   // sequencer 1
   INITIAL_STEP Initialschritt:   // S1, max time T#10S, warning time T#7S
              N    #sq.init
              R    #sq.inHoming
              R    #sq.running
              R    #sq.done
              R    "FG01Actors".Lasermarker.setWorkPos
              R    #qxNok
              R    "FG01Actors".Camera.setTrigger
   END_STEP
   TRANSITION Automatikablauf FROM Initialschritt TO Grundstellung   // T1
      := NOT #signals.isHoming;
   END_TRANSITION
   TRANSITION Grundstellungsfahrt FROM Initialschritt TO "Start Grundstellungsfahrt"   // T5
      := #signals.isHoming;
   END_TRANSITION
   STEP Grundstellung:   // S2, max time T#10S, warning time T#7S
              N    #sq.isWaiting
              N    "FG01Globals".SQ1.readyForIndex
   END_STEP
   TRANSITION Freigabe FROM Grundstellung TO SK_läuft   // T2
      := #sq.inHome AND NOT #signals.isInAutoStoping AND #sq.start AND NOT #sq.done AND #signals.releaseNextJog;
   END_TRANSITION
   STEP SK_läuft:   // S3, max time T#10S, warning time T#7S
              S    #sq.running
   END_STEP
   TRANSITION Trans3 FROM SK_läuft TO ReaderWindowToWork   // T3
      := "AlwaysTRUE";
   END_TRANSITION
   STEP Fertigmeldung:   // S4, max time T#10S, warning time T#7S
              R    #sq.running
              S    #sq.done
   END_STEP
   TRANSITION Fertig FROM Fertigmeldung TO Ende   // T4
      := "AlwaysTRUE";
   END_TRANSITION
   STEP "Start Grundstellungsfahrt":   // S5, max time T#10S, warning time T#7S
              S    #sq.inHoming
   END_STEP
   TRANSITION GST_Aktiv FROM "Start Grundstellungsfahrt" TO GS_GripperHome   // T6
      := #signals.releaseCycle;
   END_TRANSITION
   STEP "Fertig Grundstellungsfahrt":   // S6, max time T#10S, warning time T#7S
              R    #sq.inHoming
   END_STEP
   TRANSITION GST_Beendet FROM "Fertig Grundstellungsfahrt" TO Ende   // T7
      := "AlwaysTRUE";
   END_TRANSITION
   STEP Ende:   // S7, max time T#10S, warning time T#7S
   END_STEP
   TRANSITION Beendet FROM Ende TO Grundstellung   // T8, jump
      := "AlwaysTRUE";
   END_TRANSITION
   STEP ResetRelease:   // S8, max time T#10S, warning time T#7S
      supervision V := (#ResetRelease.U >= t#10s) AND NOT #DoneToIndexer.TT AND #signals.releaseCycle;
          S1  R    "TransportGlobals".Index01.release
   END_STEP
   TRANSITION DoneToIndexer FROM ResetRelease TO JogS7   // T9
      := true;
   END_TRANSITION
   STEP GS_GripperHome:   // S14, max time T#10S, warning time T#7S
      supervision V := #sstReleaseCycle.T >= #itMaxRuntime;
              R    "FG01Actors".Gripper.setWorkPos
              S    "FG01Actors".Gripper.setHomePos
   END_STEP
   TRANSITION GS_GripperInHome FROM GS_GripperHome TO GS_PlattformHome   // T15
      := "FG01Actors".Gripper.inHomePos;
   END_TRANSITION
   STEP GS_PlattformHome:   // S15, max time T#10S, warning time T#7S
      supervision V := #sstReleaseCycle.T >= #itMaxRuntime;
              S    "FG01Actors".Plattform.setHomePos
              R    "FG01Actors".Plattform.setWorkPos
   END_STEP
   TRANSITION GS_PlattformInHome FROM GS_PlattformHome TO GS_ReaderWindowHome   // T16
      := "FG01Actors".Plattform.inHomePos;
   END_TRANSITION
   STEP GS_ReaderWindowHome:   // S16, max time T#10S, warning time T#7S
      supervision V := #sstReleaseCycle.T >= #itMaxRuntime;
              R    "FG01Actors".ReaderWindow.setWorkPos
              S    "FG01Actors".ReaderWindow.setHomePos
   END_STEP
   TRANSITION GS_ReaderWindowInHome FROM GS_ReaderWindowHome TO GS_OpenGates   // T17
      := "FG01Actors".ReaderWindow.inHomePos;
   END_TRANSITION
   STEP PlattformToWork:   // S17, max time T#10S, warning time T#7S
      supervision V := #sstReleaseCycle.T >= #itMaxRuntime;
              R    "FG01Actors".Plattform.setHomePos
              S    "FG01Actors".Plattform.setWorkPos
   END_STEP
   TRANSITION PlattformIsInWork FROM PlattformToWork TO JogS4   // T18
      := "FG01Actors".Plattform.inWorkPos;
   END_TRANSITION
   STEP ReaderWindowToWork:   // S18, max time T#10S, warning time T#7S
      supervision V := #sstReleaseCycle.T >= #itMaxRuntime;
              S    "FG01Actors".ReaderWindow.setWorkPos
              R    "FG01Actors".ReaderWindow.setHomePos
   END_STEP
   TRANSITION ReaderWindowInWork FROM ReaderWindowToWork TO JogS1   // T19
      := "FG01Actors".ReaderWindow.inWorkPos;
   END_TRANSITION
   STEP GripperToWork:   // S19, max time T#10S, warning time T#7S
      supervision V := #sstReleaseCycle.T >= #itMaxRuntime;
              S    "FG01Actors".Gripper.setWorkPos
              R    "FG01Actors".Gripper.setHomePos
   END_STEP
   TRANSITION GripperInWork FROM GripperToWork TO JogS3   // T20
      := "FG01Actors".Gripper.inWorkPos;
   END_TRANSITION
   STEP GripperToHome:   // S20, max time T#10S, warning time T#7S
      supervision V := #sstReleaseCycle.T >= #itMaxRuntime;
              R    "FG01Actors".Gripper.setWorkPos
              S    "FG01Actors".Gripper.setHomePos
   END_STEP
   TRANSITION GripperInHome FROM GripperToHome TO JogS9   // T21
      := "FG01Actors".Gripper.inHomePos;
   END_TRANSITION
   STEP PlattformToHome:   // S21, max time T#10S, warning time T#7S
      supervision V := #sstReleaseCycle.T >= #itMaxRuntime;
              S    "FG01Actors".Plattform.setHomePos
              R    "FG01Actors".Plattform.setWorkPos
   END_STEP
   TRANSITION PlattformIsInWork_1 FROM PlattformToHome TO JogS8   // T22
      := "FG01Actors".Plattform.inHomePos;
   END_TRANSITION
   STEP JogS3:   // S28, max time T#10S, warning time T#7S
              N    #sq.jogDone
   END_STEP
   TRANSITION JogT3 FROM JogS3 TO PlattformToWork   // T30
      := #signals.releaseNextJog;
   END_TRANSITION
   STEP JogS4:   // S29, max time T#10S, warning time T#7S
              N    #sq.jogDone
   END_STEP
   TRANSITION JogT4 FROM JogS4 TO CheckLaserOn   // T31
      := #signals.releaseNextJog;
   END_TRANSITION
   STEP JogS1:   // S30, max time T#10S, warning time T#7S
              N    #sq.jogDone
   END_STEP
   TRANSITION JogT1 FROM JogS1 TO Set_Trigger   // T32
      := #signals.releaseNextJog;
   END_TRANSITION
   STEP JogS7:   // S31, max time T#10S, warning time T#7S
              N    #sq.jogDone
   END_STEP
   TRANSITION JogT7 FROM JogS7 TO PlattformToHome   // T33
      := #signals.releaseNextJog;
   END_TRANSITION
   STEP Laser:   // S32, max time T#10S, warning time T#7S
      supervision V := #sstReleaseCycle.T >= #itMaxRuntime;
              N    "FG01Actors".Lasermarker.setWorkPos
   END_STEP
   TRANSITION LaserDone FROM Laser TO JogS6   // T34
      := (#Laser.T >= t#3s) AND "FG01Actors".Lasermarker.workAct;
   END_TRANSITION
   STEP JogS8:   // S33, max time T#10S, warning time T#7S
              N    #sq.jogDone
   END_STEP
   TRANSITION JogT8 FROM JogS8 TO GripperToHome   // T35
      := #signals.releaseNextJog;
   END_TRANSITION
   STEP ReaderWindowToHome:   // S22, max time T#10S, warning time T#7S
      supervision V := #sstReleaseCycle.T >= #itMaxRuntime;
              R    "FG01Actors".ReaderWindow.setWorkPos
              S    "FG01Actors".ReaderWindow.setHomePos
   END_STEP
   TRANSITION ReaderWindowInHome FROM ReaderWindowToHome TO Fertigmeldung   // T23
      := "FG01Actors".ReaderWindow.inHomePos;
   END_TRANSITION
   STEP CloseGates:   // S34, max time T#10S, warning time T#7S
      supervision V := #sstReleaseCycle.T >= #itMaxRuntime;
              S    "FG01Actors".Gate_1.setWorkPos
              S    "FG01Actors".Gate_2.setWorkPos
   END_STEP
   TRANSITION GatesClosed FROM CloseGates TO JogS5   // T36
      := "FG01Actors".Gate_1.inWorkPos AND "FG01Actors".Gate_2.inWorkPos;
   END_TRANSITION
   STEP JogS5:   // S35, max time T#10S, warning time T#7S
              N    #sq.jogDone
   END_STEP
   TRANSITION JogT5 FROM JogS5 TO Laser   // T37
      := #signals.releaseNextJog;
   END_TRANSITION
   STEP JogS9:   // S36, max time T#10S, warning time T#7S
              N    #sq.jogDone
   END_STEP
   TRANSITION JogT9 FROM JogS9 TO ReaderWindowToHome   // T38
      := #signals.releaseNextJog;
   END_TRANSITION
   STEP OpenGates:   // S37, max time T#10S, warning time T#7S
      supervision V := #sstReleaseCycle.T >= #itMaxRuntime;
              R    "FG01Actors".Gate_1.setWorkPos
              R    "FG01Actors".Gate_2.setWorkPos
   END_STEP
   TRANSITION GatesOpened FROM OpenGates TO ResetRelease   // T39
      := "FG01Actors".Gate_1.inHomePos AND "FG01Actors".Gate_2.inHomePos;
   END_TRANSITION
   STEP JogS6:   // S38, max time T#10S, warning time T#7S
              N    #sq.jogDone
   END_STEP
   TRANSITION JogT6 FROM JogS6 TO OpenGates   // T40
      := #signals.releaseNextJog;
   END_TRANSITION
   STEP GS_OpenGates:   // S39, max time T#10S, warning time T#7S
      supervision V := #sstReleaseCycle.T >= #itMaxRuntime;
              R    "FG01Actors".Gate_1.setWorkPos
              R    "FG01Actors".Gate_2.setWorkPos
   END_STEP
   TRANSITION GS_GatesOpened FROM GS_OpenGates TO "Fertig Grundstellungsfahrt"   // T41
      := "FG01Actors".Gate_1.inHomePos AND "FG01Actors".Gate_2.inHomePos;
   END_TRANSITION
   STEP CheckLaserOn:   // S40, max time T#10S, warning time T#7S
   END_STEP
   TRANSITION LaserIsOn FROM CheckLaserOn TO CloseGates   // T42
      := "FG01Globals".laserOn;
   END_TRANSITION
   TRANSITION LaserIsOff FROM CheckLaserOn TO ResetRelease   // T43
      := NOT "FG01Globals".laserOn;
   END_TRANSITION
   STEP Set_Trigger:   // S9, max time T#10S, warning time T#7S
      supervision V := #sstReleaseCycle.T >= #itMaxRuntime;
              S    "FG01Actors".Camera.setTrigger
   END_STEP
   TRANSITION TriggerIsSet FROM Set_Trigger TO Wait_Busy_Done   // T10
      := "FG01Actors".Camera.isBusy;
   END_TRANSITION
   STEP Wait_Busy_Done:   // S11, max time T#10S, warning time T#7S
      supervision V := #sstReleaseCycle.T >= #itMaxRuntime;
   END_STEP
   TRANSITION CamIsDone FROM Wait_Busy_Done TO Check_Result   // T12
      := NOT "FG01Actors".Camera.isBusy;
   END_TRANSITION
   STEP Reset_Trigger:   // S12, max time T#10S, warning time T#7S
      supervision V := #sstReleaseCycle.T >= #itMaxRuntime;
              R    "FG01Actors".Camera.setTrigger
   END_STEP
   TRANSITION TriggerIsReseted FROM Reset_Trigger TO JogS2   // T13
      := "FG01Actors".Camera.isReady;
   END_TRANSITION
   STEP JogS2:   // S41, max time T#10S, warning time T#7S
              N    #sq.jogDone
   END_STEP
   TRANSITION JogT2 FROM JogS2 TO GripperToWork   // T44
      := #signals.releaseNextJog;
   END_TRANSITION
   STEP Check_Result:   // S42, max time T#10S, warning time T#7S
      supervision V := #sstReleaseCycle.T >= #itMaxRuntime;
   END_STEP
   TRANSITION "Result Ok" FROM Check_Result TO Reset_Trigger   // T45
      := "FG01Actors".Camera.resultOk;
   END_TRANSITION
   TRANSITION "Result Nok" FROM Check_Result TO NIO   // T46
      := "FG01Actors".Camera.resultNok;
   END_TRANSITION
   STEP NIO:   // S43, max time T#10S, warning time T#7S
          S1  S    #qxNok
              R    "FG01Actors".Camera.setTrigger
   END_STEP
   TRANSITION NIO_Quittiert FROM NIO TO Reset_Trigger   // T47
      := NOT #qxNok;
   END_TRANSITION

   // permanent post-instructions
   NETWORK 1
   TITLE = Störungssignal weitergeben / Forward fault signal
      #sq.error := #ERR_FLT;
   NETWORK 2
   TITLE = Ablauf ist aktiv / Sequence active
      #qxIsActive := #sq.running;
   NETWORK 3
   TITLE = steht in Grundstellung / in home position
      #qxIsInHome := #sq.inHome AND NOT #sq.running;
   NETWORK 4
   TITLE = NIO-Erkennung zurücksetzen / Reset NOK detection
      IF #signals.ack THEN #qxNok := FALSE; END_IF;
END_FUNCTION_BLOCK

FUNCTION "FG01StepSequences" : Void   // FC1110, FBD
TITLE = Schrittkettensteuerung / Sequence control
{ S7_Optimized_Access := 'TRUE' }
VERSION : 0.1
// Ersteller: Andreas Fast Automation
// Kontakt per LinkedIn: https://www.linkedin.com/in/automation-fast-andreas/
// 
// Das Projekt dient zu Demonstrationszwecken und kann frei genutzt werden.
// 
// Bausteinbeschreibung:
// Author: Andreas Fast Automation
// Kontakt per LinkedIn: https://www.linkedin.com/in/automation-fast-andreas/
// 
// This project is intended for demonstration purposes and may be used freely.
// 
// Block description:
   VAR_IN_OUT
      station : "typeStation";
   END_VAR
   VAR_TEMP
      tempInit : Bool;
      tempAck : Bool;
      tempSwAuto : Bool;
      tempSwMan : Bool;
      tempSwTap : Bool;
      tempPush : Bool;
   END_VAR
BEGIN

REGION Network 1: GRAPH-Parameter / GRAPH parameters
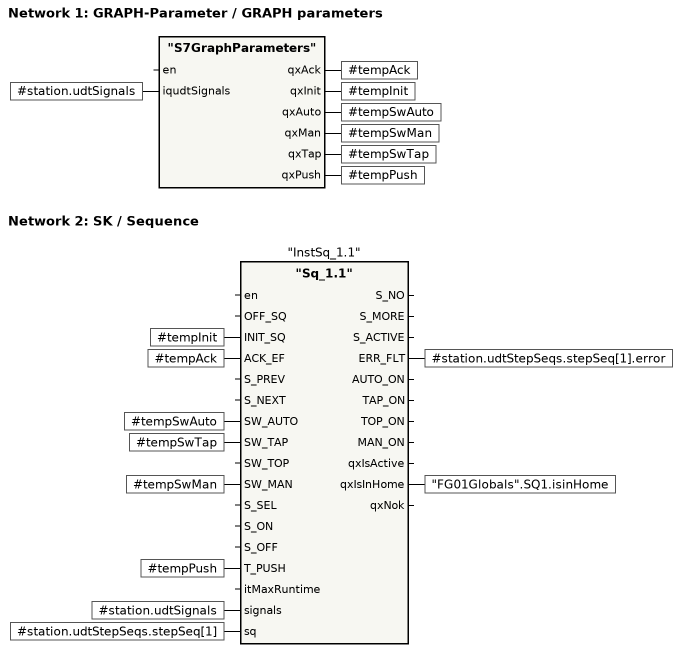
   "S7GraphParameters"(iqudtSignals := #station.udtSignals,
                       qxAck => #tempAck,
                       qxInit => #tempInit,
                       qxAuto => #tempSwAuto,
                       qxMan => #tempSwMan,
                       qxTap => #tempSwTap,
                       qxPush => #tempPush);
END_REGION

REGION Network 2: SK / Sequence
   "InstSq_1.1"(INIT_SQ := #tempInit,   // "Sq_1.1"
                ACK_EF := #tempAck,
                SW_AUTO := #tempSwAuto,
                SW_TAP := #tempSwTap,
                SW_MAN := #tempSwMan,
                T_PUSH := #tempPush,
                signals := #station.udtSignals,
                sq := #station.udtStepSeqs.stepSeq[1],
                ERR_FLT => #station.udtStepSeqs.stepSeq[1].error,
                qxIsInHome => "FG01Globals".SQ1.isinHome);
END_REGION
END_FUNCTION

// folder: 2. Machine/02_FG02

FUNCTION_BLOCK "FG02Control"   // FB1200, FBD
TITLE = Station 2 Hauptaufruf / Station 2 main call
{ S7_Optimized_Access := 'TRUE' }
VERSION : 0.1
// Ersteller: Andreas Fast Automation
// Kontakt per LinkedIn: https://www.linkedin.com/in/automation-fast-andreas/
// 
// Das Projekt dient zu Demonstrationszwecken und kann frei genutzt werden.
// 
// Bausteinbeschreibung:
// Author: Andreas Fast Automation
// Kontakt per LinkedIn: https://www.linkedin.com/in/automation-fast-andreas/
// 
// This project is intended for demonstration purposes and may be used freely.
// 
// Block description:
   VAR_INPUT
      stationNo : Int := 2;   // Stationsnummer / Station number
   END_VAR
   VAR_IN_OUT
      machine : "typeMachine";
      station : "typeStation";
      manualMovement : "typeManualMovements";
      plcErrMsg : "typePlcErrMsg";
      hmiErrMsg : "typeHmiErrMsg";
   END_VAR
   VAR
      instStationControl : "StationControl";
      instActorControl : "FG02ActorControl";
      instStationState : "StationState";
      sinstStationCycleTime : "StationCycleTime";
   END_VAR
BEGIN

REGION Network 1: Stationssteuerung / Station control
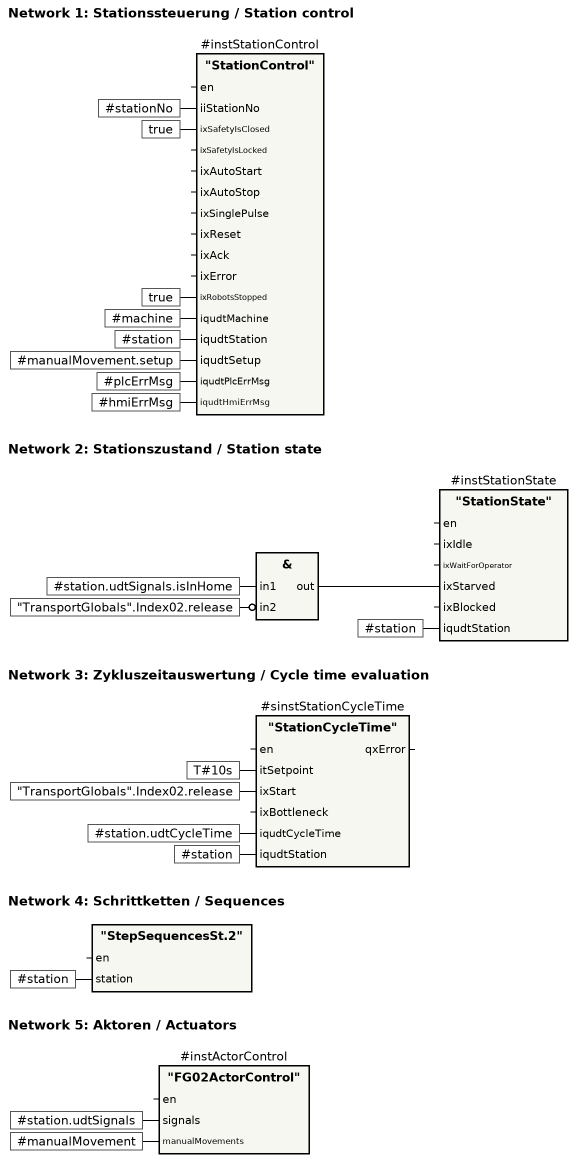
   #instStationControl(iiStationNo := #stationNo,   // "StationControl"
                       ixSafetyIsClosed := true,
                       ixRobotsStopped := true,
                       iqudtMachine := #machine,
                       iqudtStation := #station,
                       iqudtSetup := #manualMovement.setup,
                       iqudtPlcErrMsg := #plcErrMsg,
                       iqudtHmiErrMsg := #hmiErrMsg);
END_REGION

REGION Network 2: Stationszustand / Station state
   #instStationState(ixStarved := #station.udtSignals.isInHome AND NOT "TransportGlobals".Index02.release,   // "StationState"
                     iqudtStation := #station);
END_REGION

REGION Network 3: Zykluszeitauswertung / Cycle time evaluation
   #sinstStationCycleTime(itSetpoint := T#10s,   // "StationCycleTime"
                          ixStart := "TransportGlobals".Index02.release,
                          iqudtCycleTime := #station.udtCycleTime,
                          iqudtStation := #station);
END_REGION

REGION Network 4: Schrittketten / Sequences
   "StepSequencesSt.2"(station := #station);
END_REGION

REGION Network 5: Aktoren / Actuators
   #instActorControl(signals := #station.udtSignals, manualMovements := #manualMovement);   // "FG02ActorControl"
END_REGION
END_FUNCTION_BLOCK

FUNCTION_BLOCK "FG02ActorControl"   // FB1202, FBD
TITLE = Aktoransteuerung / Actuator control
{ S7_Optimized_Access := 'TRUE' }
VERSION : 0.1
// Ersteller: Andreas Fast Automation
// Kontakt per LinkedIn: https://www.linkedin.com/in/automation-fast-andreas/
// 
// Das Projekt dient zu Demonstrationszwecken und kann frei genutzt werden.
// 
// Bausteinbeschreibung:
// Author: Andreas Fast Automation
// Kontakt per LinkedIn: https://www.linkedin.com/in/automation-fast-andreas/
// 
// This project is intended for demonstration purposes and may be used freely.
// 
// Block description:
   VAR_IN_OUT
      signals : "typeStationSignals";
      manualMovements : "typeManualMovements";
   END_VAR
   VAR
      instCamera : "Actor_1Out_SimpleCamera";
      instActorReserved3 : "Actor_Reserved";
      instActorReserved4 : "Actor_Reserved";
   END_VAR
BEGIN

REGION Network 1: Kamera / Camera
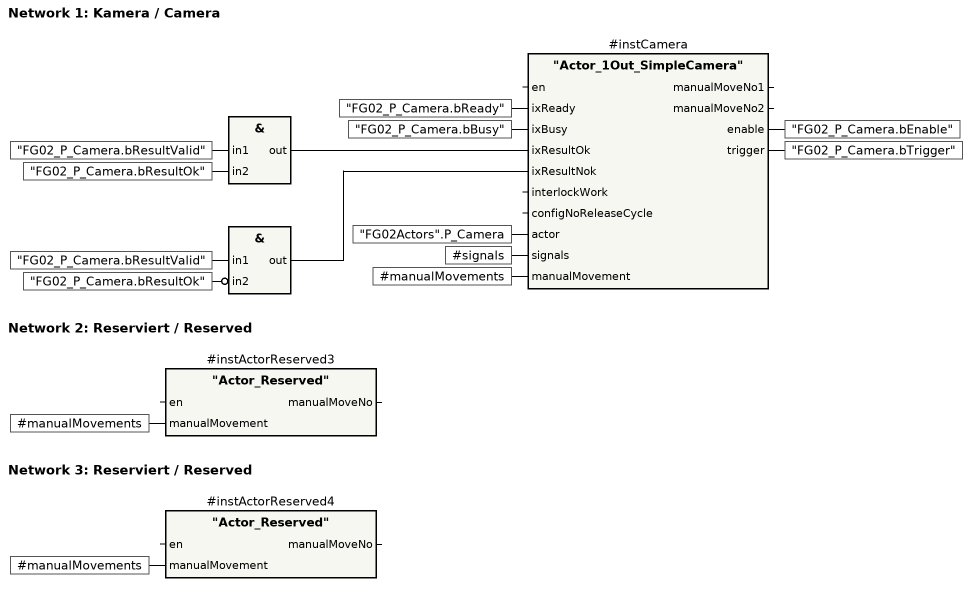
   #instCamera(ixReady := "FG02_P_Camera.bReady",   // "Actor_1Out_SimpleCamera"
               ixBusy := "FG02_P_Camera.bBusy",
               ixResultOk := "FG02_P_Camera.bResultValid" AND "FG02_P_Camera.bResultOk",
               ixResultNok := "FG02_P_Camera.bResultValid" AND NOT "FG02_P_Camera.bResultOk",
               actor := "FG02Actors".P_Camera,
               signals := #signals,
               manualMovement := #manualMovements,
               enable => "FG02_P_Camera.bEnable",
               trigger => "FG02_P_Camera.bTrigger");
END_REGION

REGION Network 2: Reserviert / Reserved
   #instActorReserved3(manualMovement := #manualMovements);   // "Actor_Reserved"
END_REGION

REGION Network 3: Reserviert / Reserved
   #instActorReserved4(manualMovement := #manualMovements);   // "Actor_Reserved"
END_REGION
END_FUNCTION_BLOCK

// folder: 2. Machine/02_FG02/Stepsequences

FUNCTION_BLOCK "Sq_2.1"   // FB1211, GRAPH_PLUS
{ S7_Optimized_Access := 'TRUE' }
VERSION : 0.1
   VAR_INPUT
      OFF_SQ : Bool := false;   // Kette ausschalten
      INIT_SQ : Bool := false;   // Kette in Initialzustand versetzen
      ACK_EF : Bool := false;   // Alle Fehler und Störungen quittieren
      S_PREV : Bool := false;   // Vorherigen Schritt am Parameter S_NO ausgeben
      S_NEXT : Bool := false;   // Nächsten Schritt am Parameter S_NO anzeigen
      SW_AUTO : Bool := false;   // Automatischer Betrieb
      SW_TAP : Bool := false;   // Halbautomatisch/Weiterschalten mit Transition
      SW_TOP : Bool := false;   // Halbautomatisch/Ignoriere Transition
      SW_MAN : Bool := false;   // Handbetrieb
      S_SEL : Int := 0;   // Schritt auswählen, der an S_NO ausgegeben werden soll
      S_ON : Bool := false;   // Schritt aktivieren, der an Parameter S_NO anliegt
      S_OFF : Bool := false;   // Schritt deaktivieren, der an Parameter S_NO anliegt
      T_PUSH : Bool := false;   // Schaltfreigabe für Transition im halbautomatischen Betrieb
      itMaxRuntime : Time := t#10s;   // Maximale Laufzeit für diesen Prozess / Maximum execution time for this process
   END_VAR
   VAR_OUTPUT
      S_NO : Int := 0;   // Schrittnummer
      S_MORE : Bool := false;   // Weitere Schritte sind vorhanden und können in S_NO angezeigt werden.
      S_ACTIVE : Bool := false;   // Schritt, der an Parameter S_NO angezeigt wird, ist aktiv
      ERR_FLT : Bool := false;   // Sammelfehler Interlock oder Supervision
      AUTO_ON : Bool := false;   // Automatischer Betrieb eingeschaltet
      TAP_ON : Bool := false;   // Halbautomatischer Betrieb/Schritt mit Transition eingeschaltet
      TOP_ON : Bool := false;   // Halbautomatischer Betrieb/Ignoriere Transition eingeschaltet
      MAN_ON : Bool := false;   // Handbetrieb eingeschaltet
      qxIsActive : Bool;   // Schrittkette läuft / Sequence running
      qxIsInHome : Bool;   // steht in Grundstellung / in home position
      qxNok : Bool;   // NIO Teil / NOK part
   END_VAR
   VAR_IN_OUT
      signals : "typeStationSignals";   // Stationssteuersignale / Station control signals
      sq : "typeStepSequence";   // Schrittkettensteuersignale / Sequence control signals
   END_VAR
   VAR
      sstReleaseCycle : Struct
         ErrorAck : Bool;
         No_LastCycle : Int;
         T : Time;   // Aktive Zeit des ReleaseCycle / Active time of ReleaseCycle
         Tck : Time;
         TckPrev : Time;
      END_STRUCT;
      HMI_INFO : Array[0..8] of UInt;
      IF_PAR : G7_IfParPlus_V6;
      RT_DATA : G7_RTDataPlus_V6;   // Interner Datenbereich
      Automatikablauf : G7_TransitionPlus_V6;   // Transitionsstruktur
      Freigabe : G7_TransitionPlus_V6;   // Transitionsstruktur
      GreiferLeer : G7_TransitionPlus_V6;   // Transitionsstruktur
      Fertig : G7_TransitionPlus_V6;   // Transitionsstruktur
      Grundstellungsfahrt : G7_TransitionPlus_V6;   // Transitionsstruktur
      GST_Aktiv : G7_TransitionPlus_V6;   // Transitionsstruktur
      GST_Beendet : G7_TransitionPlus_V6;   // Transitionsstruktur
      Beendet : G7_TransitionPlus_V6;   // Transitionsstruktur
      DoneToIndexer : G7_TransitionPlus_V6;   // Transitionsstruktur / Transition structure
      TriggerIsSet : G7_TransitionPlus_V6;   // Transitionsstruktur / Transition structure
      GS_ResetTrigger : G7_TransitionPlus_V6;   // Transition structure / Transitionsstruktur
      CamIsDone : G7_TransitionPlus_V6;   // Transition structure / Transitionsstruktur
      TriggerIsReseted : G7_TransitionPlus_V6;   // Transition structure / Transitionsstruktur
      JogT1 : G7_TransitionPlus_V6;   // Transition structure / Transitionsstruktur
      "Result Ok" : G7_TransitionPlus_V6;   // Transition structure / Transitionsstruktur
      "Result Nok" : G7_TransitionPlus_V6;   // Transition structure / Transitionsstruktur
      NIO_Quittiert : G7_TransitionPlus_V6;   // Transition structure / Transitionsstruktur
      Initialschritt : G7_StepPlus_V6;   // Schrittstruktur
      Grundstellung : G7_StepPlus_V6;   // Schrittstruktur
      SK_läuft : G7_StepPlus_V6;   // Schrittstruktur
      Fertigmeldung : G7_StepPlus_V6;   // Schrittstruktur
      "Start Grundstellungsfahrt" : G7_StepPlus_V6;   // Schrittstruktur
      "Fertig Grundstellungsfahrt" : G7_StepPlus_V6;   // Schrittstruktur
      Ende : G7_StepPlus_V6;   // Schrittstruktur
      ResetRelease : G7_StepPlus_V6;   // Schrittstruktur / Step structure
      Set_Trigger : G7_StepPlus_V6;   // Schrittstruktur / Step structure
      GS_Reset_Trigger : G7_StepPlus_V6;   // Step structure / Schrittstruktur
      Wait_Busy_Done : G7_StepPlus_V6;   // Step structure / Schrittstruktur
      Reset_Trigger : G7_StepPlus_V6;   // Step structure / Schrittstruktur
      JogS1 : G7_StepPlus_V6;   // Step structure / Schrittstruktur
      Check_Result : G7_StepPlus_V6;   // Step structure / Schrittstruktur
      NIO : G7_StepPlus_V6;   // Step structure / Schrittstruktur
      SINI : Array[0..1] of USInt;
      LSTT : Array[0..16] of USInt;
      ATAJ : Array[0..16] of USInt;
      ATAB : Array[0..16] of USInt;
      PSTT : Array[0..16] of USInt;
      NSTT : Array[0..16] of USInt;
      ASSJ : Array[0..14] of USInt;
      ASSB : Array[0..14] of USInt;
      PTTS : Array[0..14] of USInt;
      NTTS : Array[0..14] of USInt;
      SW_SQTS : Array[0..14] of USInt;
      SWITCH : Array[0..4] of USInt;
      TVX : Array[0..5] of USInt;
      TTX : Array[0..5] of USInt;
      TSX : Array[0..1] of USInt;
      S00X : Array[0..1] of USInt;
      SOFFX : Array[0..1] of USInt;
      SONX : Array[0..1] of USInt;
      SAX : Array[0..1] of USInt;
      SERRX : Array[0..15] of USInt;
      SMX : Array[0..15] of USInt;
      S0X : Array[0..15] of USInt;
      S1X : Array[0..15] of USInt;
      IL_ALARM_INST : Diag_Alarm;
      SUP_ALARM_INST : Diag_Alarm;
      STEP_TIME_ALARM_INST : Diag_Alarm;
      IEC_TIMER_INST : IEC_TIMER;
      TRANSACTION_FLAG : Bool := false;
   END_VAR
   VAR_TEMP
      txStartCondition : Bool;
      tdTckDiff : DInt;
   END_VAR
   VAR_TEMP   // added for the SCL form of the ladder/FBD networks
      _w1 : Bool;
      _w2 : Bool;
   END_VAR
   // SINI[0] := 2;
   // LSTT[0] := 255;
   // LSTT[1] := 255;
   // LSTT[2] := 255;
   // LSTT[3] := 255;
   // LSTT[4] := 255;
   // LSTT[5] := 255;
   // LSTT[6] := 255;
   // LSTT[7] := 1;
   // ATAJ[1] := 1;
   // ATAJ[2] := 2;
   // ATAJ[3] := 6;
   // ATAJ[4] := 4;
   // ATAJ[5] := 5;
   // ATAJ[6] := 3;
   // ATAJ[7] := 7;
   // ATAB[0] := 4;
   // ATAB[1] := 1;
   // ATAB[2] := 2;
   // ATAB[3] := 3;
   // ATAB[5] := 5;
   // ATAB[6] := 6;
   // ATAB[7] := 7;
   // PSTT[1] := 1;
   // PSTT[2] := 2;
   // PSTT[3] := 3;
   // PSTT[5] := 4;
   // PSTT[6] := 5;
   // PSTT[7] := 6;
   // NSTT[0] := 1;
   // NSTT[1] := 2;
   // NSTT[2] := 8;
   // NSTT[3] := 6;
   // NSTT[4] := 4;
   // NSTT[5] := 9;
   // NSTT[6] := 6;
   // NSTT[7] := 1;
   // ASSJ[1] := 1;
   // ASSJ[2] := 2;
   // ASSJ[3] := 3;
   // ASSJ[4] := 4;
   // ASSJ[5] := 5;
   // ASSJ[6] := 6;
   // ASSB[1] := 1;
   // ASSB[2] := 2;
   // ASSB[3] := 3;
   // ASSB[4] := 4;
   // ASSB[5] := 5;
   // ASSB[6] := 6;
   // PTTS[0] := 255;
   // PTTS[2] := 1;
   // PTTS[3] := 8;
   // PTTS[4] := 4;
   // PTTS[5] := 10;
   // PTTS[6] := 3;
   // NTTS[1] := 1;
   // NTTS[2] := 2;
   // NTTS[3] := 3;
   // NTTS[4] := 5;
   // NTTS[5] := 6;
   // NTTS[6] := 7;
   // SW_SQTS[1] := 1;
   // SW_SQTS[2] := 1;
   // SW_SQTS[3] := 2;
   // SW_SQTS[4] := 3;
   // SW_SQTS[5] := 3;
   // SW_SQTS[6] := 4;
   // TVX[0] := 16#1;
   // TTX[0] := 16#1;
   // TSX[0] := 16#1;
   // S00X[0] := 16#1;
   // SOFFX[0] := 16#1;
   // SONX[0] := 16#1;
   // SAX[0] := 16#1;
   // SERRX[0] := 16#1;
   // SMX[0] := 16#1;
   // S0X[0] := 16#1;
   // S1X[0] := 16#1;
   // LSTT[8] := 255;
   // ATAJ[8] := 8;
   // ATAB[8] := 8;
   // PSTT[8] := 7;
   // NSTT[8] := 3;
   // ASSJ[7] := 7;
   // ASSB[7] := 7;
   // PTTS[7] := 13;
   // NTTS[7] := 8;
   // SW_SQTS[7] := 2;
   // LSTT[9] := 255;
   // ATAJ[9] := 9;
   // ATAB[9] := 9;
   // PSTT[9] := 8;
   // NSTT[9] := 10;
   // ASSJ[8] := 8;
   // ASSB[8] := 8;
   // PTTS[8] := 2;
   // NTTS[8] := 9;
   // SW_SQTS[8] := 1;
   // LSTT[10] := 255;
   // LSTT[11] := 255;
   // LSTT[12] := 255;
   // LSTT[13] := 255;
   // ATAJ[10] := 10;
   // ATAJ[11] := 11;
   // ATAJ[12] := 12;
   // ATAJ[13] := 13;
   // ATAB[10] := 10;
   // ATAB[11] := 11;
   // ATAB[12] := 12;
   // ATAB[13] := 13;
   // PSTT[10] := 9;
   // PSTT[11] := 10;
   // PSTT[12] := 11;
   // PSTT[13] := 12;
   // NSTT[10] := 5;
   // NSTT[11] := 13;
   // NSTT[12] := 12;
   // NSTT[13] := 7;
   // ASSJ[9] := 9;
   // ASSJ[10] := 10;
   // ASSJ[11] := 11;
   // ASSJ[12] := 12;
   // ASSB[9] := 9;
   // ASSB[10] := 10;
   // ASSB[11] := 11;
   // ASSB[12] := 12;
   // PTTS[9] := 5;
   // PTTS[10] := 9;
   // PTTS[11] := 14;
   // PTTS[12] := 12;
   // NTTS[9] := 10;
   // NTTS[10] := 11;
   // NTTS[11] := 12;
   // NTTS[12] := 13;
   // SW_SQTS[9] := 3;
   // SW_SQTS[10] := 1;
   // SW_SQTS[11] := 2;
   // SW_SQTS[12] := 2;
   // LSTT[14] := 255;
   // LSTT[15] := 255;
   // ATAJ[14] := 16;
   // ATAJ[15] := 15;
   // ATAB[14] := 15;
   // ATAB[15] := 14;
   // PSTT[14] := 13;
   // PSTT[15] := 13;
   // NSTT[14] := 11;
   // NSTT[15] := 14;
   // ASSJ[13] := 13;
   // ASSB[13] := 13;
   // PTTS[13] := 11;
   // NTTS[13] := 14;
   // SW_SQTS[13] := 1;
   // LSTT[16] := 255;
   // ATAJ[16] := 14;
   // ATAB[16] := 16;
   // PSTT[16] := 14;
   // NSTT[16] := 11;
   // ASSJ[14] := 14;
   // ASSB[14] := 14;
   // PTTS[14] := 15;
   // NTTS[14] := 16;
   // SW_SQTS[14] := 5;
BEGIN
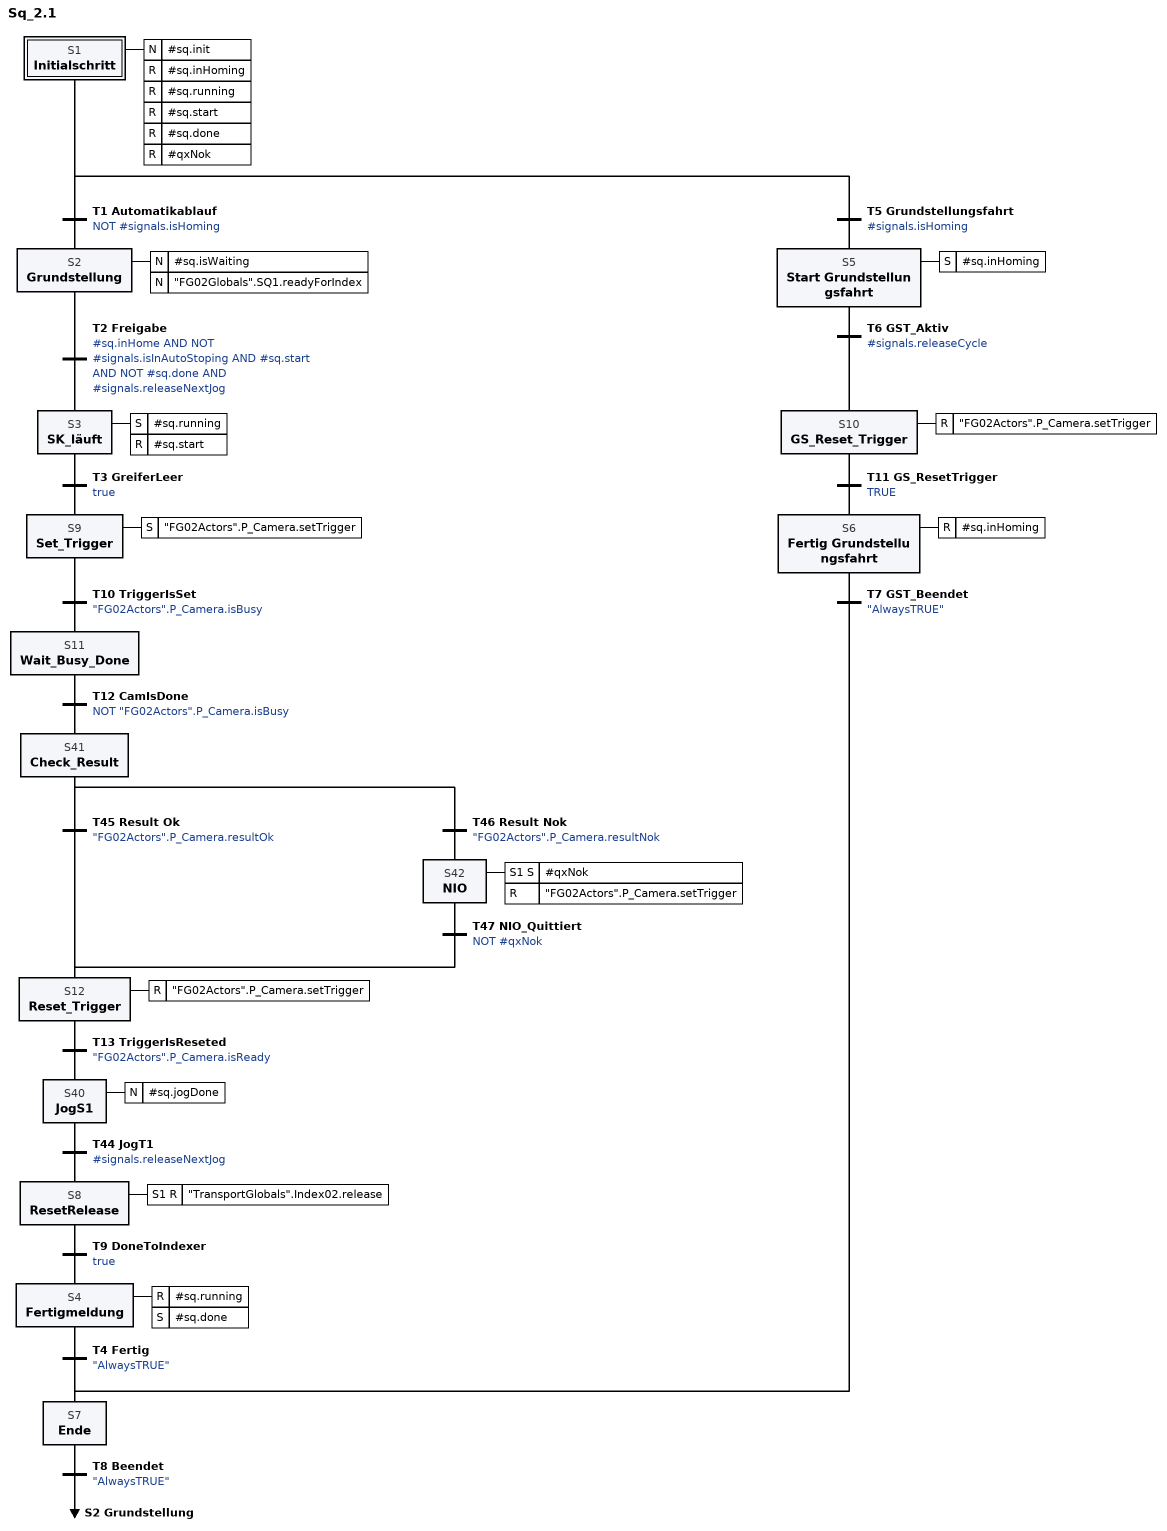
   // permanent pre-instructions
   NETWORK 1
   TITLE = Schrittkette verfügbar / Sequence available
      #sq.exists := true;
   NETWORK 2
   TITLE = Schrittkette in Grundstellung / Sequence in home position
      #sq.inHome := #Grundstellung.X AND "FG02Actors".P_Camera.isReady;
   NETWORK 3
   TITLE = Startbedingung (Erweitern) / Start condition (extend)
      #txStartCondition := "TransportGlobals".Index02.release;
   NETWORK 4
   TITLE = Schrittkette starten / Start sequence
      IF #sq.inHome AND NOT #sq.running AND #signals.releaseCycle AND NOT #signals.isHoming AND #txStartCondition THEN
          #sq.start := TRUE;
          #sq.done := FALSE;
      END_IF;
   NETWORK 5
   TITLE = ReleaseCycle-Zeitgeber / ReleaseCycle timer
      // ENO of a box is taken as its EN; it also drops when the box reports an error
      #_w1 := #ERR_FLT AND #ACK_EF;
      #_w2 := #_w1 AND NOT #sstReleaseCycle.ErrorAck;   // rising edge
      #sstReleaseCycle.ErrorAck := #_w1;
      IF (#S_NO <> #sstReleaseCycle.No_LastCycle) OR #_w2 THEN
          #sstReleaseCycle.T := T#0MS;
          #sstReleaseCycle.TckPrev := #sstReleaseCycle.Tck;
          #sstReleaseCycle.No_LastCycle := #S_NO;
      END_IF;
      #sstReleaseCycle.Tck := TIME_TCK();
      #tdTckDiff := #sstReleaseCycle.Tck - #sstReleaseCycle.TckPrev;
      #sstReleaseCycle.TckPrev := #sstReleaseCycle.Tck;
      IF (0 <= #tdTckDiff) AND (#tdTckDiff <= 1000) AND #signals.releaseCycle THEN
          #sstReleaseCycle.T := #sstReleaseCycle.T + #tdTckDiff;
      END_IF;

   // sequencer 1
   INITIAL_STEP Initialschritt:   // S1, max time T#10S, warning time T#7S
              N    #sq.init
              R    #sq.inHoming
              R    #sq.running
              R    #sq.start
              R    #sq.done
              R    #qxNok
   END_STEP
   TRANSITION Automatikablauf FROM Initialschritt TO Grundstellung   // T1
      := NOT #signals.isHoming;
   END_TRANSITION
   TRANSITION Grundstellungsfahrt FROM Initialschritt TO "Start Grundstellungsfahrt"   // T5
      := #signals.isHoming;
   END_TRANSITION
   STEP Grundstellung:   // S2, max time T#10S, warning time T#7S
      supervision V := (#Grundstellung.U > t#5S) AND NOT #sq.inHome AND #signals.releaseCycle;
              N    #sq.isWaiting
              N    "FG02Globals".SQ1.readyForIndex
   END_STEP
   TRANSITION Freigabe FROM Grundstellung TO SK_läuft   // T2
      := #sq.inHome AND NOT #signals.isInAutoStoping AND #sq.start AND NOT #sq.done AND #signals.releaseNextJog;
   END_TRANSITION
   STEP SK_läuft:   // S3, max time T#10S, warning time T#7S
              S    #sq.running
              R    #sq.start
   END_STEP
   TRANSITION GreiferLeer FROM SK_läuft TO Set_Trigger   // T3
      := true;
   END_TRANSITION
   STEP Fertigmeldung:   // S4, max time T#10S, warning time T#7S
              R    #sq.running
              S    #sq.done
   END_STEP
   TRANSITION Fertig FROM Fertigmeldung TO Ende   // T4
      := "AlwaysTRUE";
   END_TRANSITION
   STEP "Start Grundstellungsfahrt":   // S5, max time T#10S, warning time T#7S
              S    #sq.inHoming
   END_STEP
   TRANSITION GST_Aktiv FROM "Start Grundstellungsfahrt" TO GS_Reset_Trigger   // T6
      := #signals.releaseCycle;
   END_TRANSITION
   STEP "Fertig Grundstellungsfahrt":   // S6, max time T#10S, warning time T#7S
              R    #sq.inHoming
   END_STEP
   TRANSITION GST_Beendet FROM "Fertig Grundstellungsfahrt" TO Ende   // T7
      := "AlwaysTRUE";
   END_TRANSITION
   STEP Ende:   // S7, max time T#10S, warning time T#7S
   END_STEP
   TRANSITION Beendet FROM Ende TO Grundstellung   // T8, jump
      := "AlwaysTRUE";
   END_TRANSITION
   STEP Set_Trigger:   // S9, max time T#10S, warning time T#7S
      supervision V := #sstReleaseCycle.T >= #itMaxRuntime;
              S    "FG02Actors".P_Camera.setTrigger
   END_STEP
   TRANSITION TriggerIsSet FROM Set_Trigger TO Wait_Busy_Done   // T10
      := "FG02Actors".P_Camera.isBusy;
   END_TRANSITION
   STEP ResetRelease:   // S8, max time T#10S, warning time T#7S
      supervision V := #sstReleaseCycle.T >= #itMaxRuntime;
          S1  R    "TransportGlobals".Index02.release
   END_STEP
   TRANSITION DoneToIndexer FROM ResetRelease TO Fertigmeldung   // T9
      := true;
   END_TRANSITION
   STEP GS_Reset_Trigger:   // S10, max time T#10S, warning time T#7S
              R    "FG02Actors".P_Camera.setTrigger
   END_STEP
   TRANSITION GS_ResetTrigger FROM GS_Reset_Trigger TO "Fertig Grundstellungsfahrt"   // T11
      := TRUE;
   END_TRANSITION
   STEP Wait_Busy_Done:   // S11, max time T#10S, warning time T#7S
      supervision V := #sstReleaseCycle.T >= #itMaxRuntime;
   END_STEP
   TRANSITION CamIsDone FROM Wait_Busy_Done TO Check_Result   // T12
      := NOT "FG02Actors".P_Camera.isBusy;
   END_TRANSITION
   STEP Reset_Trigger:   // S12, max time T#10S, warning time T#7S
      supervision V := #sstReleaseCycle.T >= #itMaxRuntime;
              R    "FG02Actors".P_Camera.setTrigger
   END_STEP
   TRANSITION TriggerIsReseted FROM Reset_Trigger TO JogS1   // T13
      := "FG02Actors".P_Camera.isReady;
   END_TRANSITION
   STEP JogS1:   // S40, max time T#10S, warning time T#7S
              N    #sq.jogDone
   END_STEP
   TRANSITION JogT1 FROM JogS1 TO ResetRelease   // T44
      := #signals.releaseNextJog;
   END_TRANSITION
   STEP Check_Result:   // S41, max time T#10S, warning time T#7S
      supervision V := #sstReleaseCycle.T >= #itMaxRuntime;
   END_STEP
   TRANSITION "Result Ok" FROM Check_Result TO Reset_Trigger   // T45
      := "FG02Actors".P_Camera.resultOk;
   END_TRANSITION
   TRANSITION "Result Nok" FROM Check_Result TO NIO   // T46
      := "FG02Actors".P_Camera.resultNok;
   END_TRANSITION
   STEP NIO:   // S42, max time T#10S, warning time T#7S
          S1  S    #qxNok
              R    "FG02Actors".P_Camera.setTrigger
   END_STEP
   TRANSITION NIO_Quittiert FROM NIO TO Reset_Trigger   // T47
      := NOT #qxNok;
   END_TRANSITION

   // permanent post-instructions
   NETWORK 1
   TITLE = Störungssignal weitergeben / Forward fault signal
      #sq.error := #ERR_FLT;
   NETWORK 2
   TITLE = Ablauf ist aktiv / Sequence active
      #qxIsActive := #sq.running;
   NETWORK 3
   TITLE = steht in Grundstellung / in home position
      #qxIsInHome := #sq.inHome AND NOT #sq.running;
   NETWORK 4
   TITLE = NIO-Erkennung zurücksetzen / Reset NOK detection
      IF #signals.ack THEN #qxNok := FALSE; END_IF;
END_FUNCTION_BLOCK

FUNCTION "StepSequencesSt.2" : Void   // FC1210, FBD
TITLE = Schrittkettensteuerung / Sequence control
{ S7_Optimized_Access := 'TRUE' }
VERSION : 0.1
// Ersteller: Andreas Fast Automation
// Kontakt per LinkedIn: https://www.linkedin.com/in/automation-fast-andreas/
// 
// Das Projekt dient zu Demonstrationszwecken und kann frei genutzt werden.
// 
// Bausteinbeschreibung:
// Author: Andreas Fast Automation
// Kontakt per LinkedIn: https://www.linkedin.com/in/automation-fast-andreas/
// 
// This project is intended for demonstration purposes and may be used freely.
// 
// Block description:
   VAR_IN_OUT
      station : "typeStation";
   END_VAR
   VAR_TEMP
      tempInit : Bool;
      tempAck : Bool;
      tempAuto : Bool;
      tempMan : Bool;
      tempTap : Bool;
      tempPush : Bool;
   END_VAR
BEGIN

REGION Network 1: GRAPH-Parameter / GRAPH parameters
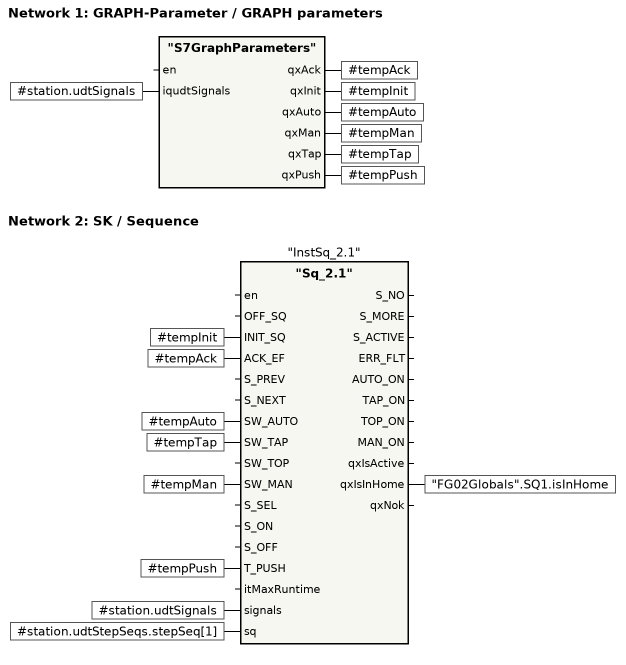
   "S7GraphParameters"(iqudtSignals := #station.udtSignals,
                       qxAck => #tempAck,
                       qxInit => #tempInit,
                       qxAuto => #tempAuto,
                       qxMan => #tempMan,
                       qxTap => #tempTap,
                       qxPush => #tempPush);
END_REGION

REGION Network 2: SK / Sequence
   "InstSq_2.1"(INIT_SQ := #tempInit,   // "Sq_2.1"
                ACK_EF := #tempAck,
                SW_AUTO := #tempAuto,
                SW_TAP := #tempTap,
                SW_MAN := #tempMan,
                T_PUSH := #tempPush,
                signals := #station.udtSignals,
                sq := #station.udtStepSeqs.stepSeq[1],
                qxIsInHome => "FG02Globals".SQ1.isInHome);
END_REGION
END_FUNCTION

// folder: 2. Machine/03_FG03

FUNCTION_BLOCK "FG03Control"   // FB1300, FBD
TITLE = Station 3 Hauptaufruf / Station 3 main call
{ S7_Optimized_Access := 'TRUE' }
VERSION : 0.1
// Ersteller: Andreas Fast Automation
// Kontakt per LinkedIn: https://www.linkedin.com/in/automation-fast-andreas/
// 
// Das Projekt dient zu Demonstrationszwecken und kann frei genutzt werden.
// 
// Bausteinbeschreibung:
// Author: Andreas Fast Automation
// Kontakt per LinkedIn: https://www.linkedin.com/in/automation-fast-andreas/
// 
// This project is intended for demonstration purposes and may be used freely.
// 
// Block description:
   VAR_INPUT
      stationNo : Int := 3;   // Stationsnummer / Station number
   END_VAR
   VAR_IN_OUT
      machine : "typeMachine";
      station : "typeStation";
      manualMovement : "typeManualMovements";
      plcErrMsg : "typePlcErrMsg";
      hmiErrMsg : "typeHmiErrMsg";
   END_VAR
   VAR
      instStationControl : "StationControl";
      instActorControl : "FG03ActorControl";
      instStationState : "StationState";
      sinstStationCycleTime : "StationCycleTime";
   END_VAR
BEGIN

REGION Network 1: Stationssteuerung / Station control
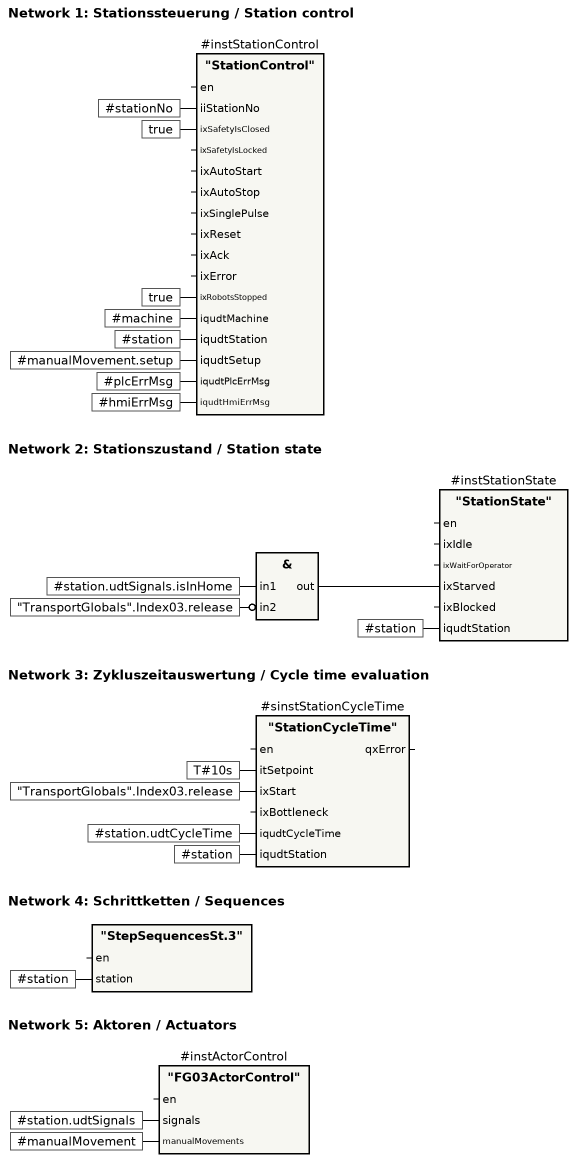
   #instStationControl(iiStationNo := #stationNo,   // "StationControl"
                       ixSafetyIsClosed := true,
                       ixRobotsStopped := true,
                       iqudtMachine := #machine,
                       iqudtStation := #station,
                       iqudtSetup := #manualMovement.setup,
                       iqudtPlcErrMsg := #plcErrMsg,
                       iqudtHmiErrMsg := #hmiErrMsg);
END_REGION

REGION Network 2: Stationszustand / Station state
   #instStationState(ixStarved := #station.udtSignals.isInHome AND NOT "TransportGlobals".Index03.release,   // "StationState"
                     iqudtStation := #station);
END_REGION

REGION Network 3: Zykluszeitauswertung / Cycle time evaluation
   #sinstStationCycleTime(itSetpoint := T#10s,   // "StationCycleTime"
                          ixStart := "TransportGlobals".Index03.release,
                          iqudtCycleTime := #station.udtCycleTime,
                          iqudtStation := #station);
END_REGION

REGION Network 4: Schrittketten / Sequences
   "StepSequencesSt.3"(station := #station);
END_REGION

REGION Network 5: Aktoren / Actuators
   #instActorControl(signals := #station.udtSignals, manualMovements := #manualMovement);   // "FG03ActorControl"
END_REGION
END_FUNCTION_BLOCK

FUNCTION_BLOCK "FG03ActorControl"   // FB1302, FBD
TITLE = Aktoransteuerung / Actuator control
{ S7_Optimized_Access := 'TRUE' }
VERSION : 0.1
// Ersteller: Andreas Fast Automation
// Kontakt per LinkedIn: https://www.linkedin.com/in/automation-fast-andreas/
// 
// Das Projekt dient zu Demonstrationszwecken und kann frei genutzt werden.
// 
// Bausteinbeschreibung:
// Author: Andreas Fast Automation
// Kontakt per LinkedIn: https://www.linkedin.com/in/automation-fast-andreas/
// 
// This project is intended for demonstration purposes and may be used freely.
// 
// Block description:
   VAR_IN_OUT
      signals : "typeStationSignals";
      manualMovements : "typeManualMovements";
   END_VAR
   VAR
      instActorReserved1 : "Actor_Reserved";
      instActorReserved2 : "Actor_Reserved";
      instActorReserved3 : "Actor_Reserved";
      instActorReserved4 : "Actor_Reserved";
      sinstAxisR1 : "Cylinder_2Out2In";
      sinstAxisX1 : "Cylinder_2Out2In";
      sinstAxisY1 : "Cylinder_2Out2In";
      sinstAxisX2 : "Cylinder_2Out2In";
      sinstAxisY2 : "Cylinder_2Out2In";
      sinstGripper1 : "Cylinder_2Out2In";
      sinstGripper2 : "Cylinder_2Out2In";
   END_VAR
BEGIN

REGION Network 1: Achse R1 / Axis R1
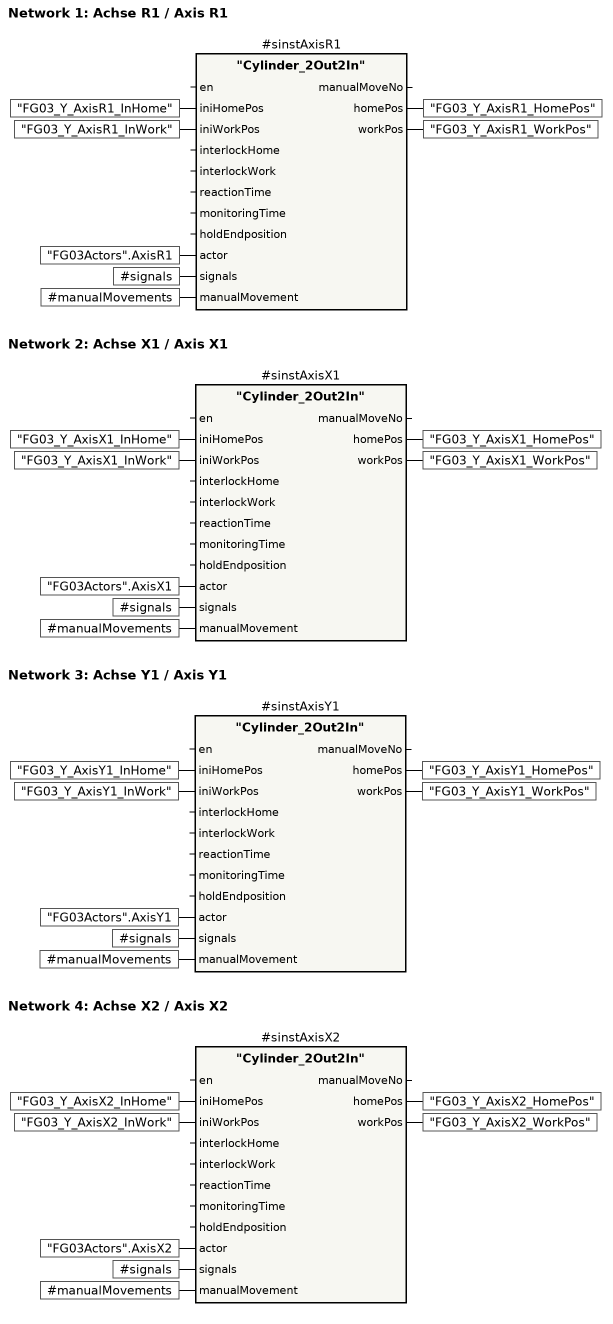
   #sinstAxisR1(iniHomePos := "FG03_Y_AxisR1_InHome",   // "Cylinder_2Out2In"
                iniWorkPos := "FG03_Y_AxisR1_InWork",
                actor := "FG03Actors".AxisR1,
                signals := #signals,
                manualMovement := #manualMovements,
                homePos => "FG03_Y_AxisR1_HomePos",
                workPos => "FG03_Y_AxisR1_WorkPos");
END_REGION

REGION Network 2: Achse X1 / Axis X1
   #sinstAxisX1(iniHomePos := "FG03_Y_AxisX1_InHome",   // "Cylinder_2Out2In"
                iniWorkPos := "FG03_Y_AxisX1_InWork",
                actor := "FG03Actors".AxisX1,
                signals := #signals,
                manualMovement := #manualMovements,
                homePos => "FG03_Y_AxisX1_HomePos",
                workPos => "FG03_Y_AxisX1_WorkPos");
END_REGION

REGION Network 3: Achse Y1 / Axis Y1
   #sinstAxisY1(iniHomePos := "FG03_Y_AxisY1_InHome",   // "Cylinder_2Out2In"
                iniWorkPos := "FG03_Y_AxisY1_InWork",
                actor := "FG03Actors".AxisY1,
                signals := #signals,
                manualMovement := #manualMovements,
                homePos => "FG03_Y_AxisY1_HomePos",
                workPos => "FG03_Y_AxisY1_WorkPos");
END_REGION

REGION Network 4: Achse X2 / Axis X2
   #sinstAxisX2(iniHomePos := "FG03_Y_AxisX2_InHome",   // "Cylinder_2Out2In"
                iniWorkPos := "FG03_Y_AxisX2_InWork",
                actor := "FG03Actors".AxisX2,
                signals := #signals,
                manualMovement := #manualMovements,
                homePos => "FG03_Y_AxisX2_HomePos",
                workPos => "FG03_Y_AxisX2_WorkPos");
END_REGION

REGION Network 5: Achse Y2 / Axis Y2
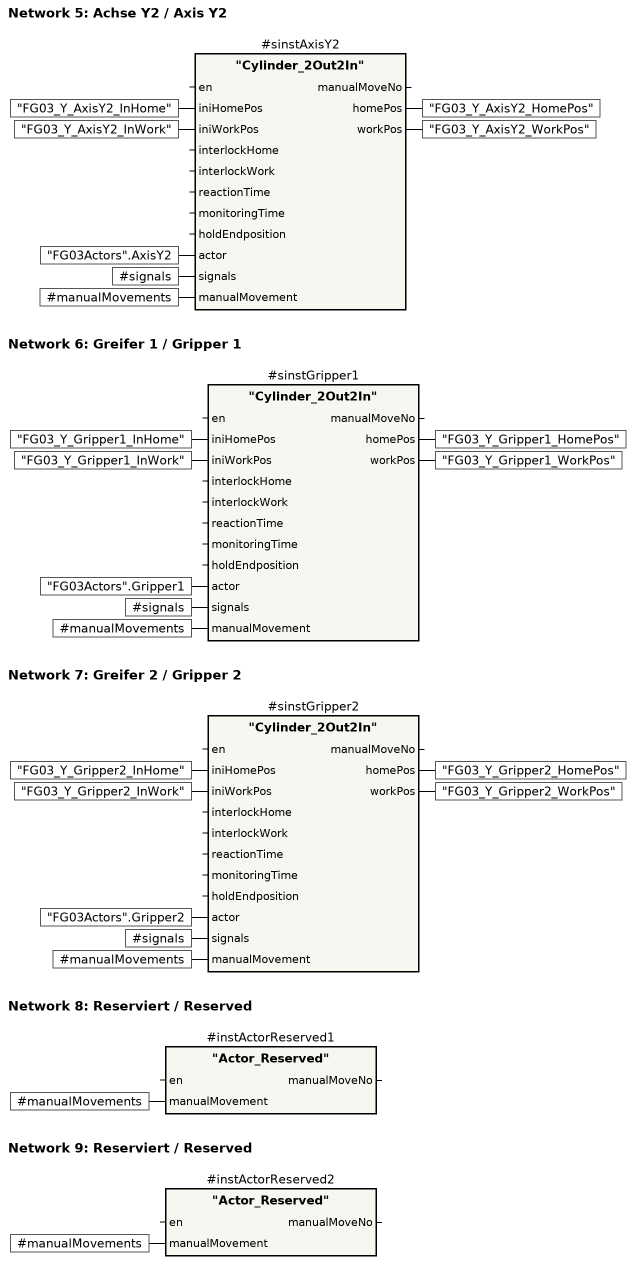
   #sinstAxisY2(iniHomePos := "FG03_Y_AxisY2_InHome",   // "Cylinder_2Out2In"
                iniWorkPos := "FG03_Y_AxisY2_InWork",
                actor := "FG03Actors".AxisY2,
                signals := #signals,
                manualMovement := #manualMovements,
                homePos => "FG03_Y_AxisY2_HomePos",
                workPos => "FG03_Y_AxisY2_WorkPos");
END_REGION

REGION Network 6: Greifer 1 / Gripper 1
   #sinstGripper1(iniHomePos := "FG03_Y_Gripper1_InHome",   // "Cylinder_2Out2In"
                  iniWorkPos := "FG03_Y_Gripper1_InWork",
                  actor := "FG03Actors".Gripper1,
                  signals := #signals,
                  manualMovement := #manualMovements,
                  homePos => "FG03_Y_Gripper1_HomePos",
                  workPos => "FG03_Y_Gripper1_WorkPos");
END_REGION

REGION Network 7: Greifer 2 / Gripper 2
   #sinstGripper2(iniHomePos := "FG03_Y_Gripper2_InHome",   // "Cylinder_2Out2In"
                  iniWorkPos := "FG03_Y_Gripper2_InWork",
                  actor := "FG03Actors".Gripper2,
                  signals := #signals,
                  manualMovement := #manualMovements,
                  homePos => "FG03_Y_Gripper2_HomePos",
                  workPos => "FG03_Y_Gripper2_WorkPos");
END_REGION

REGION Network 8: Reserviert / Reserved
   #instActorReserved1(manualMovement := #manualMovements);   // "Actor_Reserved"
END_REGION

REGION Network 9: Reserviert / Reserved
   #instActorReserved2(manualMovement := #manualMovements);   // "Actor_Reserved"
END_REGION

REGION Network 10: Reserviert / Reserved
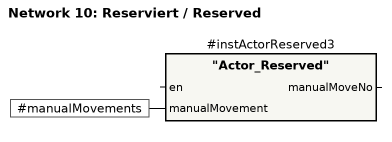
   #instActorReserved3(manualMovement := #manualMovements);   // "Actor_Reserved"
END_REGION
END_FUNCTION_BLOCK

// folder: 2. Machine/03_FG03/Stepsequences

FUNCTION_BLOCK "Sq_3.1"   // FB1311, GRAPH_PLUS
{ S7_Optimized_Access := 'TRUE' }
VERSION : 0.1
   VAR_INPUT
      OFF_SQ : Bool := false;   // Kette ausschalten
      INIT_SQ : Bool := false;   // Kette in Initialzustand versetzen
      ACK_EF : Bool := false;   // Alle Fehler und Störungen quittieren
      S_PREV : Bool := false;   // Vorherigen Schritt am Parameter S_NO ausgeben
      S_NEXT : Bool := false;   // Nächsten Schritt am Parameter S_NO anzeigen
      SW_AUTO : Bool := false;   // Automatischer Betrieb
      SW_TAP : Bool := false;   // Halbautomatisch/Weiterschalten mit Transition
      SW_TOP : Bool := false;   // Halbautomatisch/Ignoriere Transition
      SW_MAN : Bool := false;   // Handbetrieb
      S_SEL : Int := 0;   // Schritt auswählen, der an S_NO ausgegeben werden soll
      S_ON : Bool := false;   // Schritt aktivieren, der an Parameter S_NO anliegt
      S_OFF : Bool := false;   // Schritt deaktivieren, der an Parameter S_NO anliegt
      T_PUSH : Bool := false;   // Schaltfreigabe für Transition im halbautomatischen Betrieb
      itMaxRuntime : Time := t#10s;   // Maximale Laufzeit für diesen Prozess / Maximum execution time for this process
   END_VAR
   VAR_OUTPUT
      S_NO : Int := 0;   // Schrittnummer
      S_MORE : Bool := false;   // Weitere Schritte sind vorhanden und können in S_NO angezeigt werden.
      S_ACTIVE : Bool := false;   // Schritt, der an Parameter S_NO angezeigt wird, ist aktiv
      ERR_FLT : Bool := false;   // Sammelfehler Interlock oder Supervision
      AUTO_ON : Bool := false;   // Automatischer Betrieb eingeschaltet
      TAP_ON : Bool := false;   // Halbautomatischer Betrieb/Schritt mit Transition eingeschaltet
      TOP_ON : Bool := false;   // Halbautomatischer Betrieb/Ignoriere Transition eingeschaltet
      MAN_ON : Bool := false;   // Handbetrieb eingeschaltet
      qxIsActive : Bool;   // Schrittkette läuft / Sequence running
      qxIsInHome : Bool;   // steht in Grundstellung / in home position
   END_VAR
   VAR_IN_OUT
      signals : "typeStationSignals";   // Stationssteuersignale / Station control signals
      sq : "typeStepSequence";   // Schrittkettensteuersignale / Sequence control signals
   END_VAR
   VAR
      sstReleaseCycle : Struct
         ErrorAck : Bool;
         No_LastCycle : Int;
         T : Time;   // Aktive Zeit des ReleaseCycle / Active time of ReleaseCycle
         Tck : Time;
         TckPrev : Time;
      END_STRUCT;
      HMI_INFO : Array[0..8] of UInt;
      IF_PAR : G7_IfParPlus_V6;
      RT_DATA : G7_RTDataPlus_V6;   // Interner Datenbereich
      Automatikablauf : G7_TransitionPlus_V6;   // Transitionsstruktur
      Freigabe : G7_TransitionPlus_V6;   // Transitionsstruktur
      GreiferLeer : G7_TransitionPlus_V6;   // Transitionsstruktur
      Fertig : G7_TransitionPlus_V6;   // Transitionsstruktur
      Grundstellungsfahrt : G7_TransitionPlus_V6;   // Transitionsstruktur
      GST_Aktiv : G7_TransitionPlus_V6;   // Transitionsstruktur
      GST_Beendet : G7_TransitionPlus_V6;   // Transitionsstruktur
      Beendet : G7_TransitionPlus_V6;   // Transitionsstruktur
      DoneToIndexer : G7_TransitionPlus_V6;   // Transitionsstruktur / Transition structure
      GS_AxisY2InHome_1 : G7_TransitionPlus_V6;   // Transitionsstruktur / Transition structure
      GS_AxisX2InHome_1 : G7_TransitionPlus_V6;   // Transitionsstruktur / Transition structure
      GS_Gripper1InHome : G7_TransitionPlus_V6;   // Transitionsstruktur / Transition structure
      GS_AxisY2InHome_2 : G7_TransitionPlus_V6;   // Transitionsstruktur / Transition structure
      GS_AxisX2InHome_3 : G7_TransitionPlus_V6;   // Transitionsstruktur / Transition structure
      GS_AxisY2InWork : G7_TransitionPlus_V6;   // Transitionsstruktur / Transition structure
      GS_Gripper2InHome : G7_TransitionPlus_V6;   // Transitionsstruktur / Transition structure
      GS_Gripper2InHome_1 : G7_TransitionPlus_V6;   // Transitionsstruktur / Transition structure
      GS_AxisX1InHome : G7_TransitionPlus_V6;   // Transitionsstruktur / Transition structure
      GS_AxisY1InHome : G7_TransitionPlus_V6;   // Transitionsstruktur / Transition structure
      GS_AxisR1InHome : G7_TransitionPlus_V6;   // Transitionsstruktur / Transition structure
      GS_AxisR1InHome_1 : G7_TransitionPlus_V6;   // Transitionsstruktur / Transition structure
      GS_AxisX1InWork : G7_TransitionPlus_V6;   // Transitionsstruktur / Transition structure
      GS_AxisY1InWork : G7_TransitionPlus_V6;   // Transitionsstruktur / Transition structure
      GS_AxisX2InWork : G7_TransitionPlus_V6;   // Transitionsstruktur / Transition structure
      GS_Gripper2InWork : G7_TransitionPlus_V6;   // Transitionsstruktur / Transition structure
      GS_Gripper1InHome_1 : G7_TransitionPlus_V6;   // Transitionsstruktur / Transition structure
      AxisY2InWork : G7_TransitionPlus_V6;   // Transitionsstruktur / Transition structure
      JogT1 : G7_TransitionPlus_V6;   // Transitionsstruktur / Transition structure
      Gripper2InWork : G7_TransitionPlus_V6;   // Transitionsstruktur / Transition structure
      JogT2 : G7_TransitionPlus_V6;   // Transitionsstruktur / Transition structure
      AxisY2InHome : G7_TransitionPlus_V6;   // Transitionsstruktur / Transition structure
      JogT3 : G7_TransitionPlus_V6;   // Transitionsstruktur / Transition structure
      AxisX1InWork : G7_TransitionPlus_V6;   // Transitionsstruktur / Transition structure
      AxisX2InWork : G7_TransitionPlus_V6;   // Transitionsstruktur / Transition structure
      AxisY1InWork : G7_TransitionPlus_V6;   // Transitionsstruktur / Transition structure
      Gripper1InWork : G7_TransitionPlus_V6;   // Transitionsstruktur / Transition structure
      Gripper2InHome : G7_TransitionPlus_V6;   // Transitionsstruktur / Transition structure
      AxisX2InHome : G7_TransitionPlus_V6;   // Transitionsstruktur / Transition structure
      AxisR1InWork : G7_TransitionPlus_V6;   // Transitionsstruktur / Transition structure
      AxisX1InHome : G7_TransitionPlus_V6;   // Transitionsstruktur / Transition structure
      Gripper1InHome : G7_TransitionPlus_V6;   // Transitionsstruktur / Transition structure
      AxisY1InHome : G7_TransitionPlus_V6;   // Transitionsstruktur / Transition structure
      AxisR1InHome : G7_TransitionPlus_V6;   // Transitionsstruktur / Transition structure
      JogT4 : G7_TransitionPlus_V6;   // Transitionsstruktur / Transition structure
      JogT5 : G7_TransitionPlus_V6;   // Transitionsstruktur / Transition structure
      JogT6 : G7_TransitionPlus_V6;   // Transitionsstruktur / Transition structure
      JogT7 : G7_TransitionPlus_V6;   // Transitionsstruktur / Transition structure
      JogT8 : G7_TransitionPlus_V6;   // Transitionsstruktur / Transition structure
      JogT9 : G7_TransitionPlus_V6;   // Transitionsstruktur / Transition structure
      JogT10 : G7_TransitionPlus_V6;   // Transitionsstruktur / Transition structure
      JogT11 : G7_TransitionPlus_V6;   // Transitionsstruktur / Transition structure
      JogT12 : G7_TransitionPlus_V6;   // Transitionsstruktur / Transition structure
      JogT13 : G7_TransitionPlus_V6;   // Transitionsstruktur / Transition structure
      NoPartsInGripper : G7_TransitionPlus_V6;   // Transitionsstruktur / Transition structure
      PartInGripper2 : G7_TransitionPlus_V6;   // Transitionsstruktur / Transition structure
      GS_AxisY1InHome_1 : G7_TransitionPlus_V6;   // Transitionsstruktur / Transition structure
      GS_AxisY2InHome_4 : G7_TransitionPlus_V6;   // Transitionsstruktur / Transition structure
      PartInGripper1 : G7_TransitionPlus_V6;   // Transitionsstruktur / Transition structure
      GS_AxisX1InHome_1 : G7_TransitionPlus_V6;   // Transitionsstruktur / Transition structure
      GS_AxisR1InHome_2 : G7_TransitionPlus_V6;   // Transitionsstruktur / Transition structure
      GS_Gripper1InHome_2 : G7_TransitionPlus_V6;   // Transitionsstruktur / Transition structure
      Initialschritt : G7_StepPlus_V6;   // Schrittstruktur
      Grundstellung : G7_StepPlus_V6;   // Schrittstruktur
      SK_läuft : G7_StepPlus_V6;   // Schrittstruktur
      Fertigmeldung : G7_StepPlus_V6;   // Schrittstruktur
      GS_Start : G7_StepPlus_V6;   // Schrittstruktur
      "Fertig Grundstellungsfahrt" : G7_StepPlus_V6;   // Schrittstruktur
      Ende : G7_StepPlus_V6;   // Schrittstruktur
      ResetRelease : G7_StepPlus_V6;   // Schrittstruktur / Step structure
      GS_AxisY2Home_1 : G7_StepPlus_V6;   // Schrittstruktur / Step structure
      GS_AxisX2Home_1 : G7_StepPlus_V6;   // Schrittstruktur / Step structure
      GS_Gripper1Open : G7_StepPlus_V6;   // Schrittstruktur / Step structure
      GS_AxisY2Home_2 : G7_StepPlus_V6;   // Schrittstruktur / Step structure
      GS_AxisX2Home_2 : G7_StepPlus_V6;   // Schrittstruktur / Step structure
      GS_AxisY2Work : G7_StepPlus_V6;   // Schrittstruktur / Step structure
      GS_Gripper2Open : G7_StepPlus_V6;   // Schrittstruktur / Step structure
      GS_Gripper2Open_1 : G7_StepPlus_V6;   // Schrittstruktur / Step structure
      GS_AxisX1Home : G7_StepPlus_V6;   // Schrittstruktur / Step structure
      GS_AxisY1Home : G7_StepPlus_V6;   // Schrittstruktur / Step structure
      GS_AxisR1Home : G7_StepPlus_V6;   // Schrittstruktur / Step structure
      GS_AxisR1Home_1 : G7_StepPlus_V6;   // Schrittstruktur / Step structure
      GS_AxisX1Work : G7_StepPlus_V6;   // Schrittstruktur / Step structure
      GS_AxisY1Work : G7_StepPlus_V6;   // Schrittstruktur / Step structure
      GS_AxisX2Work : G7_StepPlus_V6;   // Schrittstruktur / Step structure
      GS_Gripper2Close : G7_StepPlus_V6;   // Schrittstruktur / Step structure
      GS_Gripper1Open_1 : G7_StepPlus_V6;   // Schrittstruktur / Step structure
      AxisY2Work : G7_StepPlus_V6;   // Schrittstruktur / Step structure
      JogS1 : G7_StepPlus_V6;   // Schrittstruktur / Step structure
      Gripper2Close : G7_StepPlus_V6;   // Schrittstruktur / Step structure
      JogS2 : G7_StepPlus_V6;   // Schrittstruktur / Step structure
      AxisY2Home : G7_StepPlus_V6;   // Schrittstruktur / Step structure
      JogS3 : G7_StepPlus_V6;   // Schrittstruktur / Step structure
      AxisX1Work : G7_StepPlus_V6;   // Schrittstruktur / Step structure
      AxisX2Work : G7_StepPlus_V6;   // Schrittstruktur / Step structure
      AxisY1Work : G7_StepPlus_V6;   // Schrittstruktur / Step structure
      Gripper1Close : G7_StepPlus_V6;   // Schrittstruktur / Step structure
      Gripper2Open : G7_StepPlus_V6;   // Schrittstruktur / Step structure
      AxisX2Home : G7_StepPlus_V6;   // Schrittstruktur / Step structure
      AxisR1Work : G7_StepPlus_V6;   // Schrittstruktur / Step structure
      AxisX1Home : G7_StepPlus_V6;   // Schrittstruktur / Step structure
      Gripper1Open : G7_StepPlus_V6;   // Schrittstruktur / Step structure
      AxisY1Home : G7_StepPlus_V6;   // Schrittstruktur / Step structure
      AxisR1Home : G7_StepPlus_V6;   // Schrittstruktur / Step structure
      JogS4 : G7_StepPlus_V6;   // Schrittstruktur / Step structure
      JogS5 : G7_StepPlus_V6;   // Schrittstruktur / Step structure
      JogS6 : G7_StepPlus_V6;   // Schrittstruktur / Step structure
      JogS7 : G7_StepPlus_V6;   // Schrittstruktur / Step structure
      JogS8 : G7_StepPlus_V6;   // Schrittstruktur / Step structure
      JogS9 : G7_StepPlus_V6;   // Schrittstruktur / Step structure
      JogS10 : G7_StepPlus_V6;   // Schrittstruktur / Step structure
      JogS11 : G7_StepPlus_V6;   // Schrittstruktur / Step structure
      JogS12 : G7_StepPlus_V6;   // Schrittstruktur / Step structure
      JogS13 : G7_StepPlus_V6;   // Schrittstruktur / Step structure
      GS_GripperState : G7_StepPlus_V6;   // Schrittstruktur / Step structure
      GS_AxisY2Home_4 : G7_StepPlus_V6;   // Schrittstruktur / Step structure
      GS_AxisY1Home_1 : G7_StepPlus_V6;   // Schrittstruktur / Step structure
      GS_AxisX1Home_1 : G7_StepPlus_V6;   // Schrittstruktur / Step structure
      GS_AxisR1Home_2 : G7_StepPlus_V6;   // Schrittstruktur / Step structure
      GS_Gripper1Open_2 : G7_StepPlus_V6;   // Schrittstruktur / Step structure
      SINI : Array[0..1] of USInt;
      LSTT : Array[0..60] of USInt;
      ATAJ : Array[0..60] of USInt;
      ATAB : Array[0..60] of USInt;
      PSTT : Array[0..60] of USInt;
      NSTT : Array[0..60] of USInt;
      ASSJ : Array[0..57] of USInt;
      ASSB : Array[0..57] of USInt;
      PTTS : Array[0..57] of USInt;
      NTTS : Array[0..57] of USInt;
      SW_SQTS : Array[0..57] of USInt;
      SWITCH : Array[0..6] of USInt;
      TVX : Array[0..6] of USInt;
      TTX : Array[0..6] of USInt;
      TSX : Array[0..1] of USInt;
      S00X : Array[0..1] of USInt;
      SOFFX : Array[0..1] of USInt;
      SONX : Array[0..1] of USInt;
      SAX : Array[0..1] of USInt;
      SERRX : Array[0..58] of USInt;
      SMX : Array[0..58] of USInt;
      S0X : Array[0..58] of USInt;
      S1X : Array[0..58] of USInt;
      IL_ALARM_INST : Diag_Alarm;
      SUP_ALARM_INST : Diag_Alarm;
      STEP_TIME_ALARM_INST : Diag_Alarm;
      IEC_TIMER_INST : IEC_TIMER;
      TRANSACTION_FLAG : Bool := false;
   END_VAR
   VAR_TEMP
      txStartCondition : Bool;
      tdTckDiff : DInt;
   END_VAR
   VAR_TEMP   // added for the SCL form of the ladder/FBD networks
      _w1 : Bool;
      _w2 : Bool;
   END_VAR
   // SINI[0] := 2;
   // LSTT[0] := 255;
   // LSTT[1] := 255;
   // LSTT[2] := 255;
   // LSTT[3] := 255;
   // LSTT[4] := 255;
   // LSTT[5] := 255;
   // LSTT[6] := 255;
   // LSTT[7] := 1;
   // ATAJ[1] := 1;
   // ATAJ[2] := 2;
   // ATAJ[3] := 6;
   // ATAJ[4] := 4;
   // ATAJ[5] := 5;
   // ATAJ[6] := 3;
   // ATAJ[7] := 7;
   // ATAB[0] := 4;
   // ATAB[1] := 1;
   // ATAB[2] := 2;
   // ATAB[3] := 3;
   // ATAB[5] := 5;
   // ATAB[6] := 6;
   // ATAB[7] := 7;
   // PSTT[1] := 1;
   // PSTT[2] := 2;
   // PSTT[3] := 3;
   // PSTT[5] := 4;
   // PSTT[6] := 5;
   // PSTT[7] := 6;
   // NSTT[0] := 1;
   // NSTT[1] := 2;
   // NSTT[2] := 25;
   // NSTT[3] := 6;
   // NSTT[4] := 4;
   // NSTT[5] := 52;
   // NSTT[6] := 6;
   // NSTT[7] := 1;
   // ASSJ[1] := 1;
   // ASSJ[2] := 2;
   // ASSJ[3] := 3;
   // ASSJ[4] := 4;
   // ASSJ[5] := 5;
   // ASSJ[6] := 6;
   // ASSB[1] := 1;
   // ASSB[2] := 2;
   // ASSB[3] := 3;
   // ASSB[4] := 4;
   // ASSB[5] := 5;
   // ASSB[6] := 6;
   // PTTS[0] := 255;
   // PTTS[2] := 1;
   // PTTS[3] := 42;
   // PTTS[4] := 4;
   // PTTS[5] := 19;
   // PTTS[6] := 3;
   // NTTS[1] := 1;
   // NTTS[2] := 2;
   // NTTS[3] := 3;
   // NTTS[4] := 5;
   // NTTS[5] := 6;
   // NTTS[6] := 7;
   // SW_SQTS[1] := 1;
   // SW_SQTS[2] := 1;
   // SW_SQTS[3] := 1;
   // SW_SQTS[4] := 2;
   // SW_SQTS[5] := 3;
   // SW_SQTS[6] := 4;
   // TVX[0] := 16#1;
   // TTX[0] := 16#1;
   // TSX[0] := 16#1;
   // S00X[0] := 16#1;
   // SOFFX[0] := 16#1;
   // SONX[0] := 16#1;
   // SAX[0] := 16#1;
   // SERRX[0] := 16#1;
   // SMX[0] := 16#1;
   // S0X[0] := 16#1;
   // S1X[0] := 16#1;
   // LSTT[8] := 255;
   // ATAJ[8] := 8;
   // ATAB[8] := 8;
   // PSTT[8] := 7;
   // NSTT[8] := 50;
   // ASSJ[7] := 7;
   // ASSB[7] := 7;
   // PTTS[7] := 40;
   // NTTS[7] := 8;
   // SW_SQTS[7] := 1;
   // LSTT[9] := 255;
   // ATAJ[9] := 9;
   // ATAB[9] := 9;
   // PSTT[9] := 8;
   // NSTT[9] := 9;
   // ASSJ[8] := 8;
   // ASSB[8] := 8;
   // PTTS[8] := 16;
   // NTTS[8] := 9;
   // SW_SQTS[8] := 3;
   // LSTT[10] := 255;
   // LSTT[11] := 255;
   // LSTT[12] := 255;
   // LSTT[13] := 255;
   // LSTT[14] := 255;
   // ATAJ[10] := 10;
   // ATAJ[11] := 11;
   // ATAJ[12] := 12;
   // ATAJ[13] := 13;
   // ATAJ[14] := 14;
   // ATAB[10] := 10;
   // ATAB[11] := 11;
   // ATAB[12] := 12;
   // ATAB[13] := 13;
   // ATAB[14] := 14;
   // PSTT[10] := 9;
   // PSTT[11] := 10;
   // PSTT[12] := 11;
   // PSTT[13] := 12;
   // PSTT[14] := 13;
   // NSTT[10] := 16;
   // NSTT[11] := 54;
   // NSTT[12] := 12;
   // NSTT[13] := 13;
   // NSTT[14] := 14;
   // ASSJ[9] := 9;
   // ASSJ[10] := 10;
   // ASSJ[11] := 11;
   // ASSJ[12] := 12;
   // ASSJ[13] := 13;
   // ASSB[9] := 9;
   // ASSB[10] := 10;
   // ASSB[11] := 11;
   // ASSB[12] := 12;
   // ASSB[13] := 13;
   // PTTS[9] := 9;
   // PTTS[10] := 54;
   // PTTS[11] := 59;
   // PTTS[12] := 12;
   // PTTS[13] := 13;
   // NTTS[9] := 10;
   // NTTS[10] := 11;
   // NTTS[11] := 12;
   // NTTS[12] := 13;
   // NTTS[13] := 14;
   // SW_SQTS[9] := 3;
   // SW_SQTS[10] := 5;
   // SW_SQTS[11] := 5;
   // SW_SQTS[12] := 5;
   // SW_SQTS[13] := 5;
   // LSTT[58] := 255;
   // LSTT[57] := 255;
   // LSTT[15] := 52;
   // LSTT[16] := 255;
   // LSTT[17] := 255;
   // LSTT[18] := 255;
   // LSTT[19] := 255;
   // LSTT[20] := 255;
   // LSTT[21] := 255;
   // LSTT[22] := 255;
   // LSTT[23] := 255;
   // LSTT[24] := 255;
   // LSTT[25] := 52;
   // LSTT[26] := 255;
   // LSTT[27] := 255;
   // LSTT[28] := 255;
   // LSTT[29] := 255;
   // LSTT[30] := 255;
   // ATAJ[15] := 15;
   // ATAJ[16] := 16;
   // ATAJ[17] := 17;
   // ATAJ[18] := 18;
   // ATAJ[19] := 19;
   // ATAJ[20] := 20;
   // ATAJ[21] := 21;
   // ATAJ[22] := 22;
   // ATAJ[23] := 23;
   // ATAJ[24] := 24;
   // ATAJ[25] := 25;
   // ATAJ[26] := 26;
   // ATAJ[27] := 27;
   // ATAJ[28] := 28;
   // ATAJ[29] := 29;
   // ATAJ[30] := 30;
   // ATAB[15] := 15;
   // ATAB[16] := 16;
   // ATAB[17] := 17;
   // ATAB[18] := 18;
   // ATAB[19] := 19;
   // ATAB[20] := 20;
   // ATAB[21] := 21;
   // ATAB[22] := 22;
   // ATAB[23] := 23;
   // ATAB[24] := 24;
   // ATAB[25] := 25;
   // ATAB[26] := 26;
   // ATAB[27] := 27;
   // ATAB[28] := 28;
   // ATAB[29] := 29;
   // ATAB[30] := 30;
   // PSTT[15] := 14;
   // PSTT[16] := 15;
   // PSTT[17] := 16;
   // PSTT[18] := 17;
   // PSTT[19] := 18;
   // PSTT[20] := 19;
   // PSTT[21] := 20;
   // PSTT[22] := 21;
   // PSTT[23] := 22;
   // PSTT[24] := 23;
   // PSTT[25] := 24;
   // PSTT[26] := 25;
   // PSTT[27] := 26;
   // PSTT[28] := 27;
   // PSTT[29] := 28;
   // PSTT[30] := 29;
   // NSTT[15] := 52;
   // NSTT[16] := 8;
   // NSTT[17] := 17;
   // NSTT[18] := 18;
   // NSTT[19] := 5;
   // NSTT[20] := 23;
   // NSTT[21] := 21;
   // NSTT[22] := 19;
   // NSTT[23] := 20;
   // NSTT[24] := 24;
   // NSTT[25] := 52;
   // NSTT[26] := 26;
   // NSTT[27] := 27;
   // NSTT[28] := 28;
   // NSTT[29] := 29;
   // NSTT[30] := 30;
   // ASSJ[14] := 14;
   // ASSJ[15] := 15;
   // ASSJ[16] := 16;
   // ASSJ[17] := 17;
   // ASSJ[18] := 18;
   // ASSJ[19] := 19;
   // ASSJ[20] := 20;
   // ASSJ[21] := 21;
   // ASSJ[22] := 22;
   // ASSJ[23] := 23;
   // ASSJ[24] := 24;
   // ASSJ[25] := 25;
   // ASSJ[26] := 26;
   // ASSJ[27] := 27;
   // ASSB[14] := 14;
   // ASSB[15] := 15;
   // ASSB[16] := 16;
   // ASSB[17] := 17;
   // ASSB[18] := 18;
   // ASSB[19] := 19;
   // ASSB[20] := 20;
   // ASSB[21] := 21;
   // ASSB[22] := 22;
   // ASSB[23] := 23;
   // ASSB[24] := 24;
   // ASSB[25] := 25;
   // ASSB[26] := 26;
   // ASSB[27] := 27;
   // PTTS[14] := 14;
   // PTTS[15] := 60;
   // PTTS[16] := 10;
   // PTTS[17] := 17;
   // PTTS[18] := 18;
   // PTTS[19] := 22;
   // PTTS[20] := 23;
   // PTTS[21] := 21;
   // PTTS[22] := 56;
   // PTTS[23] := 20;
   // PTTS[24] := 24;
   // PTTS[25] := 2;
   // PTTS[26] := 26;
   // PTTS[27] := 27;
   // NTTS[14] := 15;
   // NTTS[15] := 16;
   // NTTS[16] := 17;
   // NTTS[17] := 18;
   // NTTS[18] := 19;
   // NTTS[19] := 20;
   // NTTS[20] := 21;
   // NTTS[21] := 22;
   // NTTS[22] := 23;
   // NTTS[23] := 24;
   // NTTS[24] := 25;
   // NTTS[25] := 26;
   // NTTS[26] := 27;
   // NTTS[27] := 28;
   // SW_SQTS[14] := 5;
   // SW_SQTS[15] := 3;
   // SW_SQTS[16] := 3;
   // SW_SQTS[17] := 3;
   // SW_SQTS[18] := 3;
   // SW_SQTS[19] := 6;
   // SW_SQTS[20] := 6;
   // SW_SQTS[21] := 6;
   // SW_SQTS[22] := 6;
   // SW_SQTS[23] := 6;
   // SW_SQTS[24] := 6;
   // SW_SQTS[25] := 1;
   // SW_SQTS[26] := 1;
   // SW_SQTS[27] := 1;
   // LSTT[31] := 255;
   // LSTT[32] := 255;
   // LSTT[33] := 255;
   // LSTT[34] := 255;
   // LSTT[35] := 255;
   // ATAJ[31] := 31;
   // ATAJ[32] := 32;
   // ATAJ[33] := 33;
   // ATAJ[34] := 34;
   // ATAJ[35] := 35;
   // ATAB[31] := 31;
   // ATAB[32] := 32;
   // ATAB[33] := 33;
   // ATAB[34] := 34;
   // ATAB[35] := 35;
   // PSTT[31] := 30;
   // PSTT[32] := 31;
   // PSTT[33] := 32;
   // PSTT[34] := 33;
   // PSTT[35] := 34;
   // NSTT[31] := 32;
   // NSTT[32] := 43;
   // NSTT[33] := 42;
   // NSTT[34] := 44;
   // NSTT[35] := 45;
   // ASSJ[28] := 28;
   // ASSJ[29] := 29;
   // ASSJ[30] := 30;
   // ASSJ[31] := 31;
   // ASSJ[32] := 32;
   // ASSB[28] := 28;
   // ASSB[29] := 29;
   // ASSB[30] := 30;
   // ASSB[31] := 31;
   // ASSB[32] := 32;
   // PTTS[28] := 28;
   // PTTS[29] := 29;
   // PTTS[30] := 30;
   // PTTS[31] := 43;
   // PTTS[32] := 31;
   // NTTS[28] := 29;
   // NTTS[29] := 30;
   // NTTS[30] := 31;
   // NTTS[31] := 32;
   // NTTS[32] := 33;
   // SW_SQTS[28] := 1;
   // SW_SQTS[29] := 1;
   // SW_SQTS[30] := 1;
   // SW_SQTS[31] := 1;
   // SW_SQTS[32] := 1;
   // LSTT[36] := 255;
   // LSTT[37] := 255;
   // LSTT[38] := 255;
   // LSTT[39] := 255;
   // LSTT[40] := 255;
   // LSTT[41] := 255;
   // LSTT[42] := 255;
   // LSTT[43] := 255;
   // LSTT[44] := 255;
   // LSTT[45] := 255;
   // LSTT[46] := 255;
   // LSTT[47] := 255;
   // LSTT[48] := 255;
   // LSTT[49] := 255;
   // LSTT[50] := 255;
   // LSTT[51] := 255;
   // LSTT[52] := 255;
   // LSTT[53] := 255;
   // LSTT[54] := 255;
   // LSTT[55] := 255;
   // LSTT[56] := 255;
   // ATAJ[36] := 36;
   // ATAJ[37] := 37;
   // ATAJ[38] := 38;
   // ATAJ[39] := 39;
   // ATAJ[40] := 40;
   // ATAJ[41] := 41;
   // ATAJ[42] := 42;
   // ATAJ[43] := 43;
   // ATAJ[44] := 44;
   // ATAJ[45] := 45;
   // ATAJ[46] := 46;
   // ATAJ[47] := 47;
   // ATAJ[48] := 48;
   // ATAJ[49] := 49;
   // ATAJ[50] := 50;
   // ATAJ[51] := 51;
   // ATAJ[52] := 52;
   // ATAJ[53] := 53;
   // ATAJ[54] := 54;
   // ATAJ[55] := 55;
   // ATAJ[56] := 56;
   // ATAB[36] := 36;
   // ATAB[37] := 37;
   // ATAB[38] := 38;
   // ATAB[39] := 39;
   // ATAB[40] := 40;
   // ATAB[41] := 41;
   // ATAB[42] := 42;
   // ATAB[43] := 43;
   // ATAB[44] := 44;
   // ATAB[45] := 45;
   // ATAB[46] := 46;
   // ATAB[47] := 47;
   // ATAB[48] := 48;
   // ATAB[49] := 49;
   // ATAB[50] := 50;
   // ATAB[51] := 51;
   // ATAB[52] := 52;
   // ATAB[53] := 57;
   // ATAB[54] := 53;
   // ATAB[55] := 55;
   // ATAB[56] := 56;
   // PSTT[36] := 35;
   // PSTT[37] := 36;
   // PSTT[38] := 37;
   // PSTT[39] := 38;
   // PSTT[40] := 39;
   // PSTT[41] := 40;
   // PSTT[42] := 41;
   // PSTT[43] := 42;
   // PSTT[44] := 43;
   // PSTT[45] := 44;
   // PSTT[46] := 45;
   // PSTT[47] := 46;
   // PSTT[48] := 47;
   // PSTT[49] := 48;
   // PSTT[50] := 49;
   // PSTT[51] := 50;
   // PSTT[52] := 51;
   // PSTT[53] := 52;
   // PSTT[54] := 52;
   // PSTT[55] := 54;
   // PSTT[56] := 53;
   // NSTT[36] := 46;
   // NSTT[37] := 47;
   // NSTT[38] := 48;
   // NSTT[39] := 49;
   // NSTT[40] := 7;
   // NSTT[41] := 51;
   // NSTT[42] := 3;
   // NSTT[43] := 31;
   // NSTT[44] := 33;
   // NSTT[45] := 34;
   // NSTT[46] := 35;
   // NSTT[47] := 36;
   // NSTT[48] := 37;
   // NSTT[49] := 38;
   // NSTT[50] := 39;
   // NSTT[51] := 40;
   // NSTT[52] := 41;
   // NSTT[53] := 57;
   // NSTT[54] := 10;
   // NSTT[55] := 55;
   // NSTT[56] := 22;
   // ASSJ[33] := 33;
   // ASSJ[34] := 34;
   // ASSJ[35] := 35;
   // ASSJ[36] := 36;
   // ASSJ[37] := 37;
   // ASSJ[38] := 38;
   // ASSJ[39] := 39;
   // ASSJ[40] := 40;
   // ASSJ[41] := 41;
   // ASSJ[42] := 42;
   // ASSJ[43] := 43;
   // ASSJ[44] := 44;
   // ASSJ[45] := 45;
   // ASSJ[46] := 46;
   // ASSJ[47] := 47;
   // ASSJ[48] := 48;
   // ASSJ[49] := 49;
   // ASSJ[50] := 50;
   // ASSJ[51] := 51;
   // ASSJ[52] := 52;
   // ASSJ[53] := 53;
   // ASSB[33] := 33;
   // ASSB[34] := 34;
   // ASSB[35] := 35;
   // ASSB[36] := 36;
   // ASSB[37] := 37;
   // ASSB[38] := 38;
   // ASSB[39] := 39;
   // ASSB[40] := 40;
   // ASSB[41] := 41;
   // ASSB[42] := 42;
   // ASSB[43] := 43;
   // ASSB[44] := 44;
   // ASSB[45] := 45;
   // ASSB[46] := 46;
   // ASSB[47] := 47;
   // ASSB[48] := 48;
   // ASSB[49] := 49;
   // ASSB[50] := 50;
   // ASSB[51] := 51;
   // ASSB[52] := 52;
   // ASSB[53] := 53;
   // PTTS[33] := 44;
   // PTTS[34] := 45;
   // PTTS[35] := 46;
   // PTTS[36] := 47;
   // PTTS[37] := 48;
   // PTTS[38] := 49;
   // PTTS[39] := 50;
   // PTTS[40] := 51;
   // PTTS[41] := 52;
   // PTTS[42] := 33;
   // PTTS[43] := 32;
   // PTTS[44] := 34;
   // PTTS[45] := 35;
   // PTTS[46] := 36;
   // PTTS[47] := 37;
   // PTTS[48] := 38;
   // PTTS[49] := 39;
   // PTTS[50] := 8;
   // PTTS[51] := 41;
   // PTTS[52] := 5;
   // PTTS[53] := 57;
   // NTTS[33] := 34;
   // NTTS[34] := 35;
   // NTTS[35] := 36;
   // NTTS[36] := 37;
   // NTTS[37] := 38;
   // NTTS[38] := 39;
   // NTTS[39] := 40;
   // NTTS[40] := 41;
   // NTTS[41] := 42;
   // NTTS[42] := 43;
   // NTTS[43] := 44;
   // NTTS[44] := 45;
   // NTTS[45] := 46;
   // NTTS[46] := 47;
   // NTTS[47] := 48;
   // NTTS[48] := 49;
   // NTTS[49] := 50;
   // NTTS[50] := 51;
   // NTTS[51] := 52;
   // NTTS[52] := 53;
   // NTTS[53] := 56;
   // SW_SQTS[33] := 1;
   // SW_SQTS[34] := 1;
   // SW_SQTS[35] := 1;
   // SW_SQTS[36] := 1;
   // SW_SQTS[37] := 1;
   // SW_SQTS[38] := 1;
   // SW_SQTS[39] := 1;
   // SW_SQTS[40] := 1;
   // SW_SQTS[41] := 1;
   // SW_SQTS[42] := 1;
   // SW_SQTS[43] := 1;
   // SW_SQTS[44] := 1;
   // SW_SQTS[45] := 1;
   // SW_SQTS[46] := 1;
   // SW_SQTS[47] := 1;
   // SW_SQTS[48] := 1;
   // SW_SQTS[49] := 1;
   // SW_SQTS[50] := 1;
   // SW_SQTS[51] := 1;
   // SW_SQTS[52] := 2;
   // SW_SQTS[53] := 6;
   // ATAJ[57] := 57;
   // ATAJ[58] := 58;
   // ATAB[57] := 54;
   // ATAB[58] := 58;
   // PSTT[57] := 52;
   // PSTT[58] := 55;
   // NSTT[57] := 53;
   // NSTT[58] := 56;
   // ASSJ[54] := 54;
   // ASSJ[55] := 55;
   // ASSB[54] := 54;
   // ASSB[55] := 55;
   // PTTS[54] := 11;
   // PTTS[55] := 55;
   // NTTS[54] := 55;
   // NTTS[55] := 58;
   // SW_SQTS[54] := 5;
   // SW_SQTS[55] := 5;
   // LSTT[59] := 255;
   // LSTT[60] := 255;
   // ATAJ[59] := 59;
   // ATAJ[60] := 60;
   // ATAB[59] := 59;
   // ATAB[60] := 60;
   // PSTT[59] := 56;
   // PSTT[60] := 57;
   // NSTT[59] := 11;
   // NSTT[60] := 15;
   // ASSJ[56] := 56;
   // ASSJ[57] := 57;
   // ASSB[56] := 56;
   // ASSB[57] := 57;
   // PTTS[56] := 58;
   // PTTS[57] := 53;
   // NTTS[56] := 59;
   // NTTS[57] := 60;
   // SW_SQTS[56] := 5;
   // SW_SQTS[57] := 3;
BEGIN
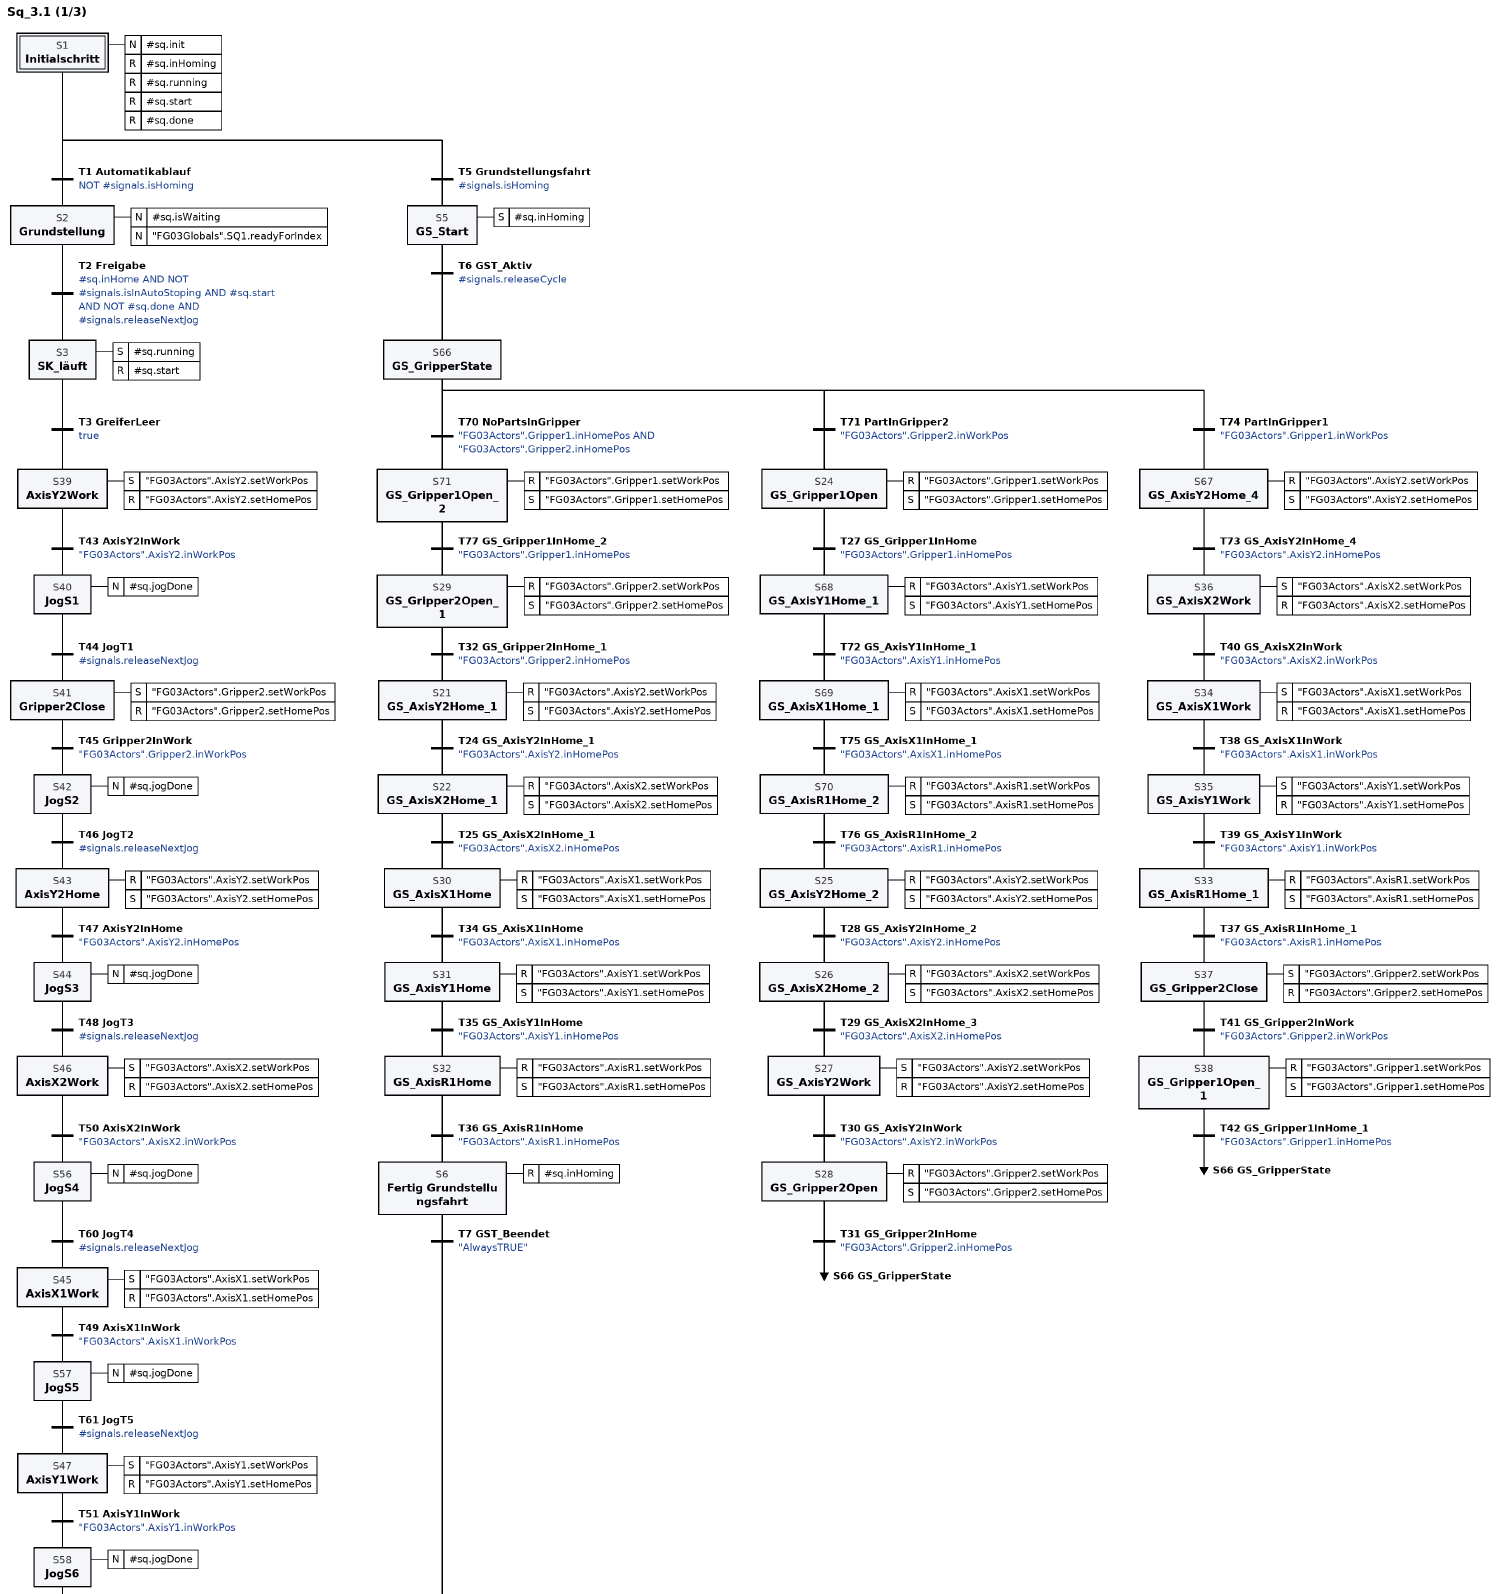
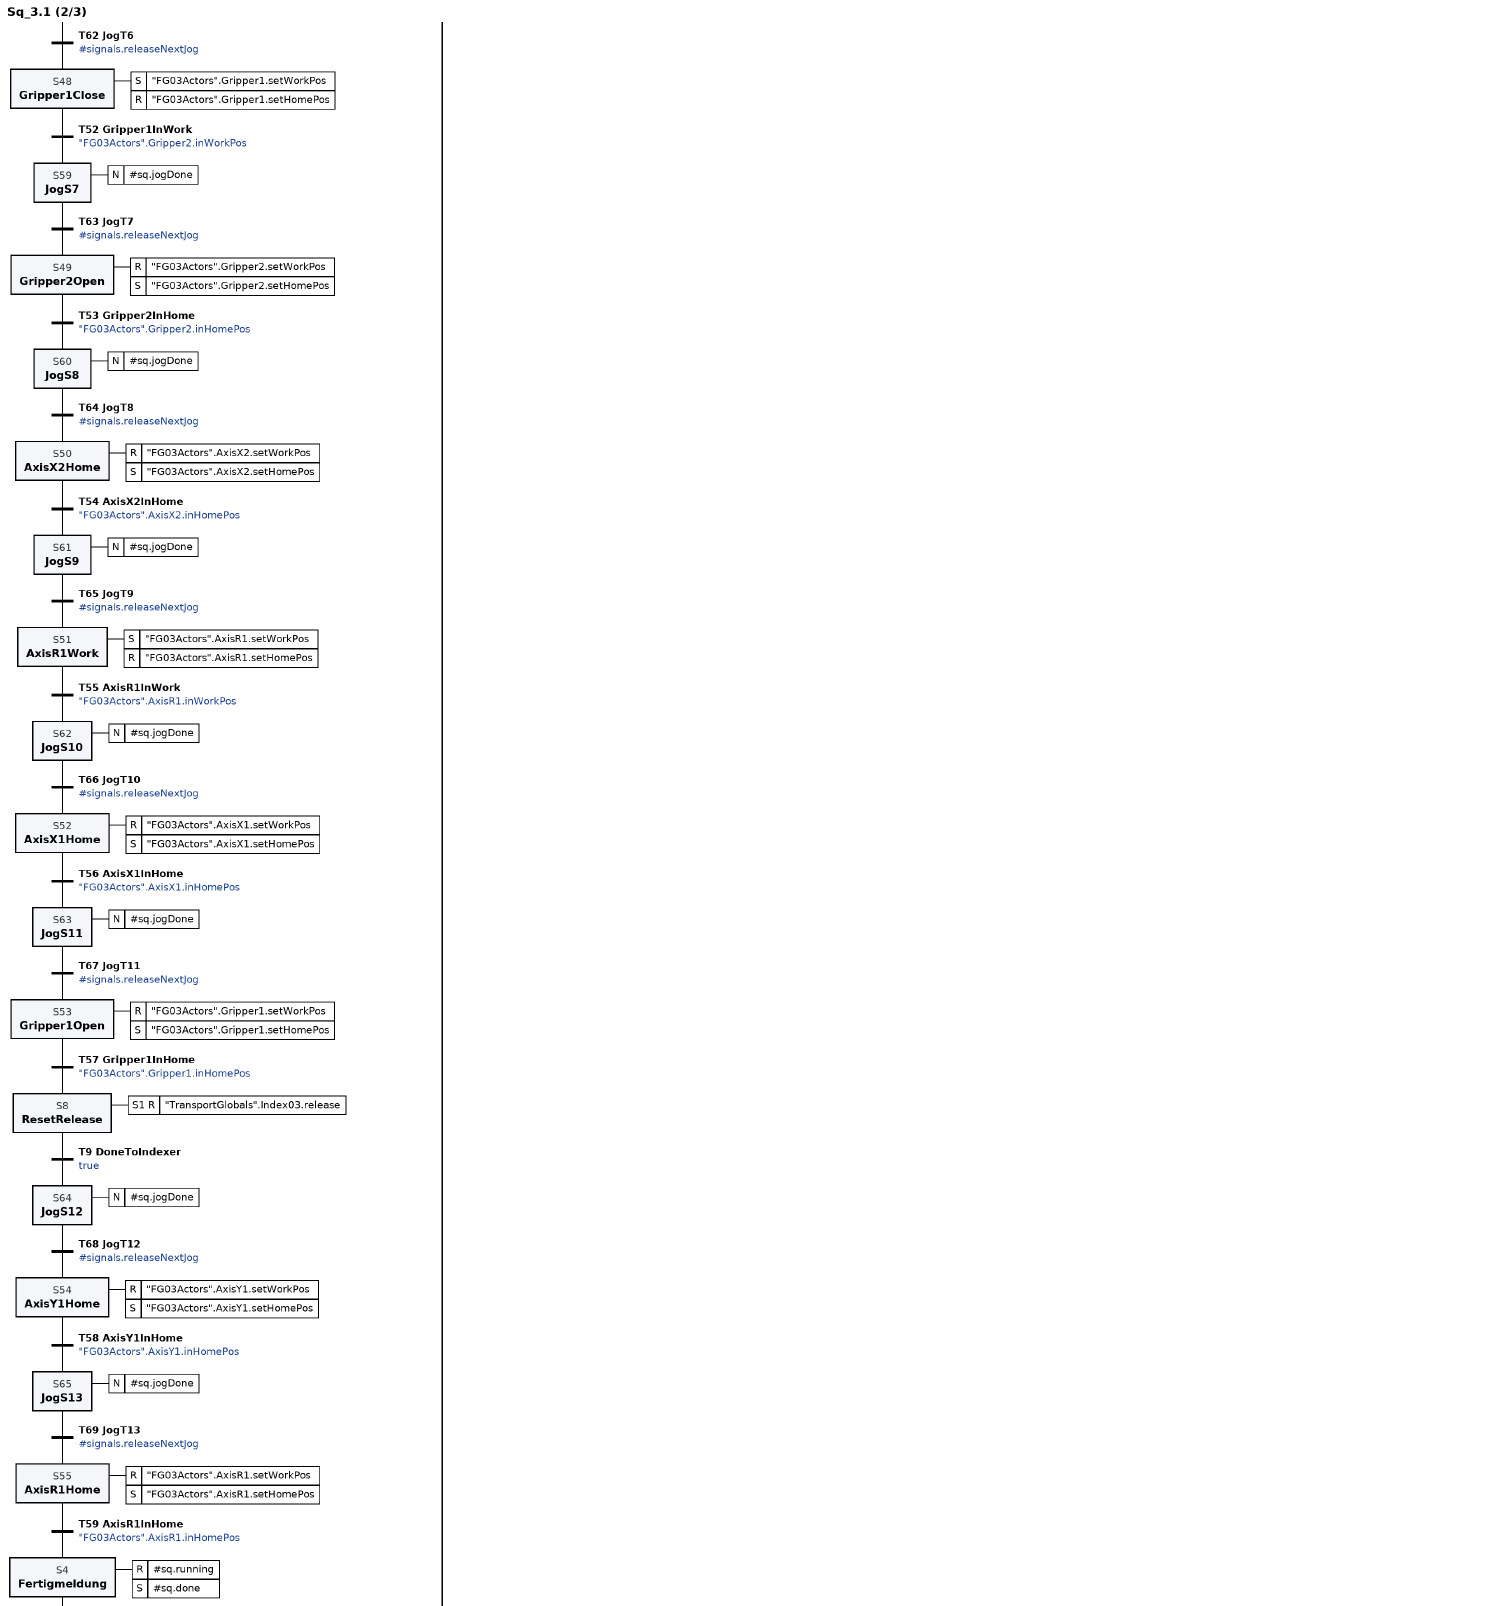
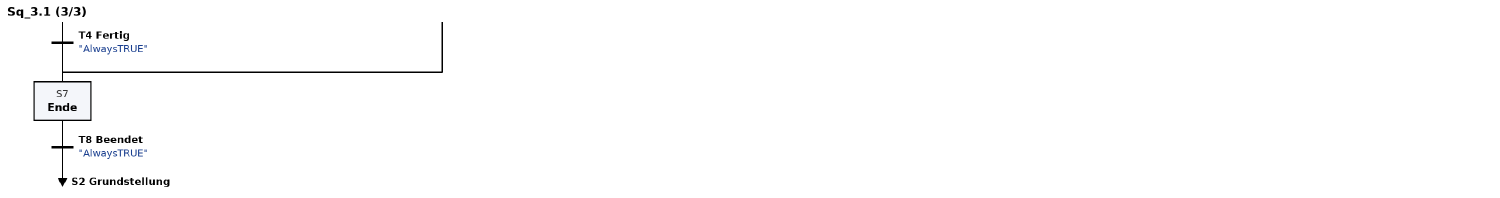
   // permanent pre-instructions
   NETWORK 1
   TITLE = Schrittkette verfügbar / Sequence available
      #sq.exists := true;
   NETWORK 2
   TITLE = Schrittkette in Grundstellung / Sequence in home position
      #sq.inHome := #Grundstellung.X AND "FG03Actors".AxisR1.inHomePos AND "FG03Actors".AxisX1.inHomePos AND "FG03Actors".AxisY1.inHomePos AND "FG03Actors".AxisX2.inHomePos AND "FG03Actors".AxisY2.inHomePos AND "FG03Actors".Gripper1.inHomePos AND "FG03Actors".Gripper2.inHomePos;
   NETWORK 3
   TITLE = Startbedingung (Erweitern) / Start condition (extend)
      #txStartCondition := "TransportGlobals".Index03.release;
   NETWORK 4
   TITLE = Schrittkette starten / Start sequence
      IF #sq.inHome AND NOT #sq.running AND #signals.releaseCycle AND NOT #signals.isHoming AND #txStartCondition THEN
          #sq.start := TRUE;
          #sq.done := FALSE;
      END_IF;
   NETWORK 5
   TITLE = ReleaseCycle-Zeitgeber / ReleaseCycle timer
      // ENO of a box is taken as its EN; it also drops when the box reports an error
      #_w1 := #ERR_FLT AND #ACK_EF;
      #_w2 := #_w1 AND NOT #sstReleaseCycle.ErrorAck;   // rising edge
      #sstReleaseCycle.ErrorAck := #_w1;
      IF (#S_NO <> #sstReleaseCycle.No_LastCycle) OR #_w2 THEN
          #sstReleaseCycle.T := T#0MS;
          #sstReleaseCycle.TckPrev := #sstReleaseCycle.Tck;
          #sstReleaseCycle.No_LastCycle := #S_NO;
      END_IF;
      #sstReleaseCycle.Tck := TIME_TCK();
      #tdTckDiff := #sstReleaseCycle.Tck - #sstReleaseCycle.TckPrev;
      #sstReleaseCycle.TckPrev := #sstReleaseCycle.Tck;
      IF (0 <= #tdTckDiff) AND (#tdTckDiff <= 1000) AND #signals.releaseCycle THEN
          #sstReleaseCycle.T := #sstReleaseCycle.T + #tdTckDiff;
      END_IF;

   // sequencer 1
   INITIAL_STEP Initialschritt:   // S1, max time T#10S, warning time T#7S
              N    #sq.init
              R    #sq.inHoming
              R    #sq.running
              R    #sq.start
              R    #sq.done
   END_STEP
   TRANSITION Automatikablauf FROM Initialschritt TO Grundstellung   // T1
      := NOT #signals.isHoming;
   END_TRANSITION
   TRANSITION Grundstellungsfahrt FROM Initialschritt TO GS_Start   // T5
      := #signals.isHoming;
   END_TRANSITION
   STEP Grundstellung:   // S2, max time T#10S, warning time T#7S
      supervision V := (#Grundstellung.U > t#5S) AND NOT #sq.inHome AND #signals.releaseCycle;
              N    #sq.isWaiting
              N    "FG03Globals".SQ1.readyForIndex
   END_STEP
   TRANSITION Freigabe FROM Grundstellung TO SK_läuft   // T2
      := #sq.inHome AND NOT #signals.isInAutoStoping AND #sq.start AND NOT #sq.done AND #signals.releaseNextJog;
   END_TRANSITION
   STEP SK_läuft:   // S3, max time T#10S, warning time T#7S
              S    #sq.running
              R    #sq.start
   END_STEP
   TRANSITION GreiferLeer FROM SK_läuft TO AxisY2Work   // T3
      := true;
   END_TRANSITION
   STEP Fertigmeldung:   // S4, max time T#10S, warning time T#7S
              R    #sq.running
              S    #sq.done
   END_STEP
   TRANSITION Fertig FROM Fertigmeldung TO Ende   // T4
      := "AlwaysTRUE";
   END_TRANSITION
   STEP GS_Start:   // S5, max time T#10S, warning time T#7S
              S    #sq.inHoming
   END_STEP
   TRANSITION GST_Aktiv FROM GS_Start TO GS_GripperState   // T6
      := #signals.releaseCycle;
   END_TRANSITION
   STEP "Fertig Grundstellungsfahrt":   // S6, max time T#10S, warning time T#7S
              R    #sq.inHoming
   END_STEP
   TRANSITION GST_Beendet FROM "Fertig Grundstellungsfahrt" TO Ende   // T7
      := "AlwaysTRUE";
   END_TRANSITION
   STEP Ende:   // S7, max time T#10S, warning time T#7S
   END_STEP
   TRANSITION Beendet FROM Ende TO Grundstellung   // T8, jump
      := "AlwaysTRUE";
   END_TRANSITION
   STEP JogS1:   // S40, max time T#10S, warning time T#7S
              N    #sq.jogDone
   END_STEP
   TRANSITION JogT1 FROM JogS1 TO Gripper2Close   // T44
      := #signals.releaseNextJog;
   END_TRANSITION
   STEP ResetRelease:   // S8, max time T#10S, warning time T#7S
      supervision V := (#ResetRelease.U >= t#10s) AND NOT #DoneToIndexer.TT AND #signals.releaseCycle;
          S1  R    "TransportGlobals".Index03.release
   END_STEP
   TRANSITION DoneToIndexer FROM ResetRelease TO JogS12   // T9
      := true;
   END_TRANSITION
   STEP GS_Gripper1Open_1:   // S38, max time T#10S, warning time T#7S
      supervision V := #sstReleaseCycle.T >= #itMaxRuntime;
              R    "FG03Actors".Gripper1.setWorkPos
              S    "FG03Actors".Gripper1.setHomePos
   END_STEP
   TRANSITION GS_Gripper1InHome_1 FROM GS_Gripper1Open_1 TO GS_GripperState   // T42, jump
      := "FG03Actors".Gripper1.inHomePos;
   END_TRANSITION
   STEP GS_AxisX2Work:   // S36, max time T#10S, warning time T#7S
      supervision V := #sstReleaseCycle.T >= #itMaxRuntime;
              S    "FG03Actors".AxisX2.setWorkPos
              R    "FG03Actors".AxisX2.setHomePos
   END_STEP
   TRANSITION GS_AxisX2InWork FROM GS_AxisX2Work TO GS_AxisX1Work   // T40
      := "FG03Actors".AxisX2.inWorkPos;
   END_TRANSITION
   STEP GS_AxisX1Work:   // S34, max time T#10S, warning time T#7S
      supervision V := #sstReleaseCycle.T >= #itMaxRuntime;
              S    "FG03Actors".AxisX1.setWorkPos
              R    "FG03Actors".AxisX1.setHomePos
   END_STEP
   TRANSITION GS_AxisX1InWork FROM GS_AxisX1Work TO GS_AxisY1Work   // T38
      := "FG03Actors".AxisX1.inWorkPos;
   END_TRANSITION
   STEP GS_AxisY2Home_4:   // S67, max time T#10S, warning time T#7S
      supervision V := #sstReleaseCycle.T >= #itMaxRuntime;
              R    "FG03Actors".AxisY2.setWorkPos
              S    "FG03Actors".AxisY2.setHomePos
   END_STEP
   TRANSITION GS_AxisY2InHome_4 FROM GS_AxisY2Home_4 TO GS_AxisX2Work   // T73
      := "FG03Actors".AxisY2.inHomePos;
   END_TRANSITION
   STEP GS_AxisR1Home_1:   // S33, max time T#10S, warning time T#7S
      supervision V := #sstReleaseCycle.T >= #itMaxRuntime;
              R    "FG03Actors".AxisR1.setWorkPos
              S    "FG03Actors".AxisR1.setHomePos
   END_STEP
   TRANSITION GS_AxisR1InHome_1 FROM GS_AxisR1Home_1 TO GS_Gripper2Close   // T37
      := "FG03Actors".AxisR1.inHomePos;
   END_TRANSITION
   STEP GS_Gripper2Close:   // S37, max time T#10S, warning time T#7S
      supervision V := #sstReleaseCycle.T >= #itMaxRuntime;
              S    "FG03Actors".Gripper2.setWorkPos
              R    "FG03Actors".Gripper2.setHomePos
   END_STEP
   TRANSITION GS_Gripper2InWork FROM GS_Gripper2Close TO GS_Gripper1Open_1   // T41
      := "FG03Actors".Gripper2.inWorkPos;
   END_TRANSITION
   STEP GS_AxisY1Home_1:   // S68, max time T#10S, warning time T#7S
      supervision V := #sstReleaseCycle.T >= #itMaxRuntime;
              R    "FG03Actors".AxisY1.setWorkPos
              S    "FG03Actors".AxisY1.setHomePos
   END_STEP
   TRANSITION GS_AxisY1InHome_1 FROM GS_AxisY1Home_1 TO GS_AxisX1Home_1   // T72
      := "FG03Actors".AxisY1.inHomePos;
   END_TRANSITION
   STEP GS_AxisY2Home_1:   // S21, max time T#10S, warning time T#7S
      supervision V := #sstReleaseCycle.T >= #itMaxRuntime;
              R    "FG03Actors".AxisY2.setWorkPos
              S    "FG03Actors".AxisY2.setHomePos
   END_STEP
   TRANSITION GS_AxisY2InHome_1 FROM GS_AxisY2Home_1 TO GS_AxisX2Home_1   // T24
      := "FG03Actors".AxisY2.inHomePos;
   END_TRANSITION
   STEP GS_AxisX2Home_1:   // S22, max time T#10S, warning time T#7S
      supervision V := #sstReleaseCycle.T >= #itMaxRuntime;
              R    "FG03Actors".AxisX2.setWorkPos
              S    "FG03Actors".AxisX2.setHomePos
   END_STEP
   TRANSITION GS_AxisX2InHome_1 FROM GS_AxisX2Home_1 TO GS_AxisX1Home   // T25
      := "FG03Actors".AxisX2.inHomePos;
   END_TRANSITION
   STEP GS_Gripper1Open:   // S24, max time T#10S, warning time T#7S
      supervision V := #sstReleaseCycle.T >= #itMaxRuntime;
              R    "FG03Actors".Gripper1.setWorkPos
              S    "FG03Actors".Gripper1.setHomePos
   END_STEP
   TRANSITION GS_Gripper1InHome FROM GS_Gripper1Open TO GS_AxisY1Home_1   // T27
      := "FG03Actors".Gripper1.inHomePos;
   END_TRANSITION
   STEP GS_AxisY2Home_2:   // S25, max time T#10S, warning time T#7S
      supervision V := #sstReleaseCycle.T >= #itMaxRuntime;
              R    "FG03Actors".AxisY2.setWorkPos
              S    "FG03Actors".AxisY2.setHomePos
   END_STEP
   TRANSITION GS_AxisY2InHome_2 FROM GS_AxisY2Home_2 TO GS_AxisX2Home_2   // T28
      := "FG03Actors".AxisY2.inHomePos;
   END_TRANSITION
   STEP GS_AxisX2Home_2:   // S26, max time T#10S, warning time T#7S
      supervision V := #sstReleaseCycle.T >= #itMaxRuntime;
              R    "FG03Actors".AxisX2.setWorkPos
              S    "FG03Actors".AxisX2.setHomePos
   END_STEP
   TRANSITION GS_AxisX2InHome_3 FROM GS_AxisX2Home_2 TO GS_AxisY2Work   // T29
      := "FG03Actors".AxisX2.inHomePos;
   END_TRANSITION
   STEP GS_AxisY2Work:   // S27, max time T#10S, warning time T#7S
      supervision V := #sstReleaseCycle.T >= #itMaxRuntime;
              S    "FG03Actors".AxisY2.setWorkPos
              R    "FG03Actors".AxisY2.setHomePos
   END_STEP
   TRANSITION GS_AxisY2InWork FROM GS_AxisY2Work TO GS_Gripper2Open   // T30
      := "FG03Actors".AxisY2.inWorkPos;
   END_TRANSITION
   STEP GS_Gripper2Open:   // S28, max time T#10S, warning time T#7S
      supervision V := #sstReleaseCycle.T >= #itMaxRuntime;
              R    "FG03Actors".Gripper2.setWorkPos
              S    "FG03Actors".Gripper2.setHomePos
   END_STEP
   TRANSITION GS_Gripper2InHome FROM GS_Gripper2Open TO GS_GripperState   // T31, jump
      := "FG03Actors".Gripper2.inHomePos;
   END_TRANSITION
   STEP GS_AxisX1Home:   // S30, max time T#10S, warning time T#7S
      supervision V := #sstReleaseCycle.T >= #itMaxRuntime;
              R    "FG03Actors".AxisX1.setWorkPos
              S    "FG03Actors".AxisX1.setHomePos
   END_STEP
   TRANSITION GS_AxisX1InHome FROM GS_AxisX1Home TO GS_AxisY1Home   // T34
      := "FG03Actors".AxisX1.inHomePos;
   END_TRANSITION
   STEP GS_AxisY1Home:   // S31, max time T#10S, warning time T#7S
      supervision V := #sstReleaseCycle.T >= #itMaxRuntime;
              R    "FG03Actors".AxisY1.setWorkPos
              S    "FG03Actors".AxisY1.setHomePos
   END_STEP
   TRANSITION GS_AxisY1InHome FROM GS_AxisY1Home TO GS_AxisR1Home   // T35
      := "FG03Actors".AxisY1.inHomePos;
   END_TRANSITION
   STEP GS_AxisR1Home:   // S32, max time T#10S, warning time T#7S
      supervision V := #sstReleaseCycle.T >= #itMaxRuntime;
              R    "FG03Actors".AxisR1.setWorkPos
              S    "FG03Actors".AxisR1.setHomePos
   END_STEP
   TRANSITION GS_AxisR1InHome FROM GS_AxisR1Home TO "Fertig Grundstellungsfahrt"   // T36
      := "FG03Actors".AxisR1.inHomePos;
   END_TRANSITION
   STEP AxisY2Work:   // S39, max time T#10S, warning time T#7S
      supervision V := #sstReleaseCycle.T >= #itMaxRuntime;
              S    "FG03Actors".AxisY2.setWorkPos
              R    "FG03Actors".AxisY2.setHomePos
   END_STEP
   TRANSITION AxisY2InWork FROM AxisY2Work TO JogS1   // T43
      := "FG03Actors".AxisY2.inWorkPos;
   END_TRANSITION
   STEP Gripper2Close:   // S41, max time T#10S, warning time T#7S
      supervision V := #sstReleaseCycle.T >= #itMaxRuntime;
              S    "FG03Actors".Gripper2.setWorkPos
              R    "FG03Actors".Gripper2.setHomePos
   END_STEP
   TRANSITION Gripper2InWork FROM Gripper2Close TO JogS2   // T45
      := "FG03Actors".Gripper2.inWorkPos;
   END_TRANSITION
   STEP JogS2:   // S42, max time T#10S, warning time T#7S
              N    #sq.jogDone
   END_STEP
   TRANSITION JogT2 FROM JogS2 TO AxisY2Home   // T46
      := #signals.releaseNextJog;
   END_TRANSITION
   STEP AxisY2Home:   // S43, max time T#10S, warning time T#7S
      supervision V := #sstReleaseCycle.T >= #itMaxRuntime;
              R    "FG03Actors".AxisY2.setWorkPos
              S    "FG03Actors".AxisY2.setHomePos
   END_STEP
   TRANSITION AxisY2InHome FROM AxisY2Home TO JogS3   // T47
      := "FG03Actors".AxisY2.inHomePos;
   END_TRANSITION
   STEP JogS3:   // S44, max time T#10S, warning time T#7S
              N    #sq.jogDone
   END_STEP
   TRANSITION JogT3 FROM JogS3 TO AxisX2Work   // T48
      := #signals.releaseNextJog;
   END_TRANSITION
   STEP AxisX1Work:   // S45, max time T#10S, warning time T#7S
      supervision V := #sstReleaseCycle.T >= #itMaxRuntime;
              S    "FG03Actors".AxisX1.setWorkPos
              R    "FG03Actors".AxisX1.setHomePos
   END_STEP
   TRANSITION AxisX1InWork FROM AxisX1Work TO JogS5   // T49
      := "FG03Actors".AxisX1.inWorkPos;
   END_TRANSITION
   STEP AxisX2Work:   // S46, max time T#10S, warning time T#7S
      supervision V := #sstReleaseCycle.T >= #itMaxRuntime;
              S    "FG03Actors".AxisX2.setWorkPos
              R    "FG03Actors".AxisX2.setHomePos
   END_STEP
   TRANSITION AxisX2InWork FROM AxisX2Work TO JogS4   // T50
      := "FG03Actors".AxisX2.inWorkPos;
   END_TRANSITION
   STEP AxisY1Work:   // S47, max time T#10S, warning time T#7S
      supervision V := #sstReleaseCycle.T >= #itMaxRuntime;
              S    "FG03Actors".AxisY1.setWorkPos
              R    "FG03Actors".AxisY1.setHomePos
   END_STEP
   TRANSITION AxisY1InWork FROM AxisY1Work TO JogS6   // T51
      := "FG03Actors".AxisY1.inWorkPos;
   END_TRANSITION
   STEP Gripper1Close:   // S48, max time T#10S, warning time T#7S
      supervision V := #sstReleaseCycle.T >= #itMaxRuntime;
              S    "FG03Actors".Gripper1.setWorkPos
              R    "FG03Actors".Gripper1.setHomePos
   END_STEP
   TRANSITION Gripper1InWork FROM Gripper1Close TO JogS7   // T52
      := "FG03Actors".Gripper2.inWorkPos;
   END_TRANSITION
   STEP Gripper2Open:   // S49, max time T#10S, warning time T#7S
      supervision V := #sstReleaseCycle.T >= #itMaxRuntime;
              R    "FG03Actors".Gripper2.setWorkPos
              S    "FG03Actors".Gripper2.setHomePos
   END_STEP
   TRANSITION Gripper2InHome FROM Gripper2Open TO JogS8   // T53
      := "FG03Actors".Gripper2.inHomePos;
   END_TRANSITION
   STEP AxisX2Home:   // S50, max time T#10S, warning time T#7S
      supervision V := #sstReleaseCycle.T >= #itMaxRuntime;
              R    "FG03Actors".AxisX2.setWorkPos
              S    "FG03Actors".AxisX2.setHomePos
   END_STEP
   TRANSITION AxisX2InHome FROM AxisX2Home TO JogS9   // T54
      := "FG03Actors".AxisX2.inHomePos;
   END_TRANSITION
   STEP AxisR1Work:   // S51, max time T#10S, warning time T#7S
      supervision V := #sstReleaseCycle.T >= #itMaxRuntime;
              S    "FG03Actors".AxisR1.setWorkPos
              R    "FG03Actors".AxisR1.setHomePos
   END_STEP
   TRANSITION AxisR1InWork FROM AxisR1Work TO JogS10   // T55
      := "FG03Actors".AxisR1.inWorkPos;
   END_TRANSITION
   STEP AxisX1Home:   // S52, max time T#10S, warning time T#7S
      supervision V := #sstReleaseCycle.T >= #itMaxRuntime;
              R    "FG03Actors".AxisX1.setWorkPos
              S    "FG03Actors".AxisX1.setHomePos
   END_STEP
   TRANSITION AxisX1InHome FROM AxisX1Home TO JogS11   // T56
      := "FG03Actors".AxisX1.inHomePos;
   END_TRANSITION
   STEP Gripper1Open:   // S53, max time T#10S, warning time T#7S
      supervision V := #sstReleaseCycle.T >= #itMaxRuntime;
              R    "FG03Actors".Gripper1.setWorkPos
              S    "FG03Actors".Gripper1.setHomePos
   END_STEP
   TRANSITION Gripper1InHome FROM Gripper1Open TO ResetRelease   // T57
      := "FG03Actors".Gripper1.inHomePos;
   END_TRANSITION
   STEP AxisY1Home:   // S54, max time T#10S, warning time T#7S
      supervision V := #sstReleaseCycle.T >= #itMaxRuntime;
              R    "FG03Actors".AxisY1.setWorkPos
              S    "FG03Actors".AxisY1.setHomePos
   END_STEP
   TRANSITION AxisY1InHome FROM AxisY1Home TO JogS13   // T58
      := "FG03Actors".AxisY1.inHomePos;
   END_TRANSITION
   STEP AxisR1Home:   // S55, max time T#10S, warning time T#7S
      supervision V := #sstReleaseCycle.T >= #itMaxRuntime;
              R    "FG03Actors".AxisR1.setWorkPos
              S    "FG03Actors".AxisR1.setHomePos
   END_STEP
   TRANSITION AxisR1InHome FROM AxisR1Home TO Fertigmeldung   // T59
      := "FG03Actors".AxisR1.inHomePos;
   END_TRANSITION
   STEP JogS4:   // S56, max time T#10S, warning time T#7S
              N    #sq.jogDone
   END_STEP
   TRANSITION JogT4 FROM JogS4 TO AxisX1Work   // T60
      := #signals.releaseNextJog;
   END_TRANSITION
   STEP JogS5:   // S57, max time T#10S, warning time T#7S
              N    #sq.jogDone
   END_STEP
   TRANSITION JogT5 FROM JogS5 TO AxisY1Work   // T61
      := #signals.releaseNextJog;
   END_TRANSITION
   STEP JogS6:   // S58, max time T#10S, warning time T#7S
              N    #sq.jogDone
   END_STEP
   TRANSITION JogT6 FROM JogS6 TO Gripper1Close   // T62
      := #signals.releaseNextJog;
   END_TRANSITION
   STEP JogS7:   // S59, max time T#10S, warning time T#7S
              N    #sq.jogDone
   END_STEP
   TRANSITION JogT7 FROM JogS7 TO Gripper2Open   // T63
      := #signals.releaseNextJog;
   END_TRANSITION
   STEP JogS8:   // S60, max time T#10S, warning time T#7S
              N    #sq.jogDone
   END_STEP
   TRANSITION JogT8 FROM JogS8 TO AxisX2Home   // T64
      := #signals.releaseNextJog;
   END_TRANSITION
   STEP JogS9:   // S61, max time T#10S, warning time T#7S
              N    #sq.jogDone
   END_STEP
   TRANSITION JogT9 FROM JogS9 TO AxisR1Work   // T65
      := #signals.releaseNextJog;
   END_TRANSITION
   STEP JogS10:   // S62, max time T#10S, warning time T#7S
              N    #sq.jogDone
   END_STEP
   TRANSITION JogT10 FROM JogS10 TO AxisX1Home   // T66
      := #signals.releaseNextJog;
   END_TRANSITION
   STEP JogS11:   // S63, max time T#10S, warning time T#7S
              N    #sq.jogDone
   END_STEP
   TRANSITION JogT11 FROM JogS11 TO Gripper1Open   // T67
      := #signals.releaseNextJog;
   END_TRANSITION
   STEP JogS12:   // S64, max time T#10S, warning time T#7S
              N    #sq.jogDone
   END_STEP
   TRANSITION JogT12 FROM JogS12 TO AxisY1Home   // T68
      := #signals.releaseNextJog;
   END_TRANSITION
   STEP JogS13:   // S65, max time T#10S, warning time T#7S
              N    #sq.jogDone
   END_STEP
   TRANSITION JogT13 FROM JogS13 TO AxisR1Home   // T69
      := #signals.releaseNextJog;
   END_TRANSITION
   STEP GS_GripperState:   // S66, max time T#10S, warning time T#7S
      supervision V := #sstReleaseCycle.T >= #itMaxRuntime;
   END_STEP
   TRANSITION NoPartsInGripper FROM GS_GripperState TO GS_Gripper1Open_2   // T70
      := "FG03Actors".Gripper1.inHomePos AND "FG03Actors".Gripper2.inHomePos;
   END_TRANSITION
   TRANSITION PartInGripper2 FROM GS_GripperState TO GS_Gripper1Open   // T71
      := "FG03Actors".Gripper2.inWorkPos;
   END_TRANSITION
   TRANSITION PartInGripper1 FROM GS_GripperState TO GS_AxisY2Home_4   // T74
      := "FG03Actors".Gripper1.inWorkPos;
   END_TRANSITION
   STEP GS_AxisY1Work:   // S35, max time T#10S, warning time T#7S
      supervision V := #sstReleaseCycle.T >= #itMaxRuntime;
              S    "FG03Actors".AxisY1.setWorkPos
              R    "FG03Actors".AxisY1.setHomePos
   END_STEP
   TRANSITION GS_AxisY1InWork FROM GS_AxisY1Work TO GS_AxisR1Home_1   // T39
      := "FG03Actors".AxisY1.inWorkPos;
   END_TRANSITION
   STEP GS_AxisX1Home_1:   // S69, max time T#10S, warning time T#7S
      supervision V := #sstReleaseCycle.T >= #itMaxRuntime;
              R    "FG03Actors".AxisX1.setWorkPos
              S    "FG03Actors".AxisX1.setHomePos
   END_STEP
   TRANSITION GS_AxisX1InHome_1 FROM GS_AxisX1Home_1 TO GS_AxisR1Home_2   // T75
      := "FG03Actors".AxisX1.inHomePos;
   END_TRANSITION
   STEP GS_AxisR1Home_2:   // S70, max time T#10S, warning time T#7S
      supervision V := #sstReleaseCycle.T >= #itMaxRuntime;
              R    "FG03Actors".AxisR1.setWorkPos
              S    "FG03Actors".AxisR1.setHomePos
   END_STEP
   TRANSITION GS_AxisR1InHome_2 FROM GS_AxisR1Home_2 TO GS_AxisY2Home_2   // T76
      := "FG03Actors".AxisR1.inHomePos;
   END_TRANSITION
   STEP GS_Gripper1Open_2:   // S71, max time T#10S, warning time T#7S
      supervision V := #sstReleaseCycle.T >= #itMaxRuntime;
              R    "FG03Actors".Gripper1.setWorkPos
              S    "FG03Actors".Gripper1.setHomePos
   END_STEP
   TRANSITION GS_Gripper1InHome_2 FROM GS_Gripper1Open_2 TO GS_Gripper2Open_1   // T77
      := "FG03Actors".Gripper1.inHomePos;
   END_TRANSITION
   STEP GS_Gripper2Open_1:   // S29, max time T#10S, warning time T#7S
      supervision V := #sstReleaseCycle.T >= #itMaxRuntime;
              R    "FG03Actors".Gripper2.setWorkPos
              S    "FG03Actors".Gripper2.setHomePos
   END_STEP
   TRANSITION GS_Gripper2InHome_1 FROM GS_Gripper2Open_1 TO GS_AxisY2Home_1   // T32
      := "FG03Actors".Gripper2.inHomePos;
   END_TRANSITION

   // permanent post-instructions
   NETWORK 1
   TITLE = Störungssignal weitergeben / Forward fault signal
      #sq.error := #ERR_FLT;
   NETWORK 2
   TITLE = Ablauf ist aktiv / Sequence active
      #qxIsActive := #sq.running;
   NETWORK 3
   TITLE = steht in Grundstellung / in home position
      #qxIsInHome := #sq.inHome AND NOT #sq.running;
END_FUNCTION_BLOCK

FUNCTION "StepSequencesSt.3" : Void   // FC1310, FBD
TITLE = Schrittkettensteuerung / Sequence control
{ S7_Optimized_Access := 'TRUE' }
VERSION : 0.1
// Ersteller: Andreas Fast Automation
// Kontakt per LinkedIn: https://www.linkedin.com/in/automation-fast-andreas/
// 
// Das Projekt dient zu Demonstrationszwecken und kann frei genutzt werden.
// 
// Bausteinbeschreibung:
// Author: Andreas Fast Automation
// Kontakt per LinkedIn: https://www.linkedin.com/in/automation-fast-andreas/
// 
// This project is intended for demonstration purposes and may be used freely.
// 
// Block description:
   VAR_IN_OUT
      station : "typeStation";
   END_VAR
   VAR_TEMP
      tempInit : Bool;
      tempAck : Bool;
      tempAuto : Bool;
      tempMan : Bool;
      tempTap : Bool;
      tempPush : Bool;
   END_VAR
BEGIN

REGION Network 1: GRAPH-Parameter / GRAPH parameters
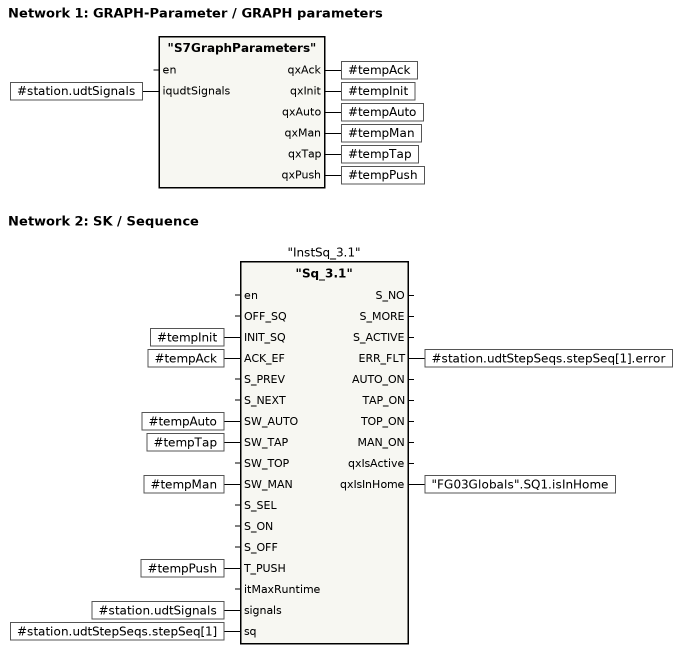
   "S7GraphParameters"(iqudtSignals := #station.udtSignals,
                       qxAck => #tempAck,
                       qxInit => #tempInit,
                       qxAuto => #tempAuto,
                       qxMan => #tempMan,
                       qxTap => #tempTap,
                       qxPush => #tempPush);
END_REGION

REGION Network 2: SK / Sequence
   "InstSq_3.1"(INIT_SQ := #tempInit,   // "Sq_3.1"
                ACK_EF := #tempAck,
                SW_AUTO := #tempAuto,
                SW_TAP := #tempTap,
                SW_MAN := #tempMan,
                T_PUSH := #tempPush,
                signals := #station.udtSignals,
                sq := #station.udtStepSeqs.stepSeq[1],
                ERR_FLT => #station.udtStepSeqs.stepSeq[1].error,
                qxIsInHome => "FG03Globals".SQ1.isInHome);
END_REGION
END_FUNCTION

// folder: 2. Machine/04_FG04

FUNCTION_BLOCK "FG04Control"   // FB1400, FBD
TITLE = Station 4 Hauptaufruf / Station 4 main call
{ S7_Optimized_Access := 'TRUE' }
VERSION : 0.1
// Ersteller: Andreas Fast Automation
// Kontakt per LinkedIn: https://www.linkedin.com/in/automation-fast-andreas/
// 
// Das Projekt dient zu Demonstrationszwecken und kann frei genutzt werden.
// 
// Bausteinbeschreibung:
// Author: Andreas Fast Automation
// Kontakt per LinkedIn: https://www.linkedin.com/in/automation-fast-andreas/
// 
// This project is intended for demonstration purposes and may be used freely.
// 
// Block description:
   VAR_INPUT
      stationNo : Int := 3;   // Stationsnummer / Station number
   END_VAR
   VAR_IN_OUT
      machine : "typeMachine";
      station : "typeStation";
      manualMovement : "typeManualMovements";
      plcErrMsg : "typePlcErrMsg";
      hmiErrMsg : "typeHmiErrMsg";
   END_VAR
   VAR
      instStationControl : "StationControl";
      instActorControl : "FG04ActorControl";
      instStationState : "StationState";
      sinstStationCycleTime : "StationCycleTime";
   END_VAR
BEGIN

REGION Network 1: Stationssteuerung / Station control
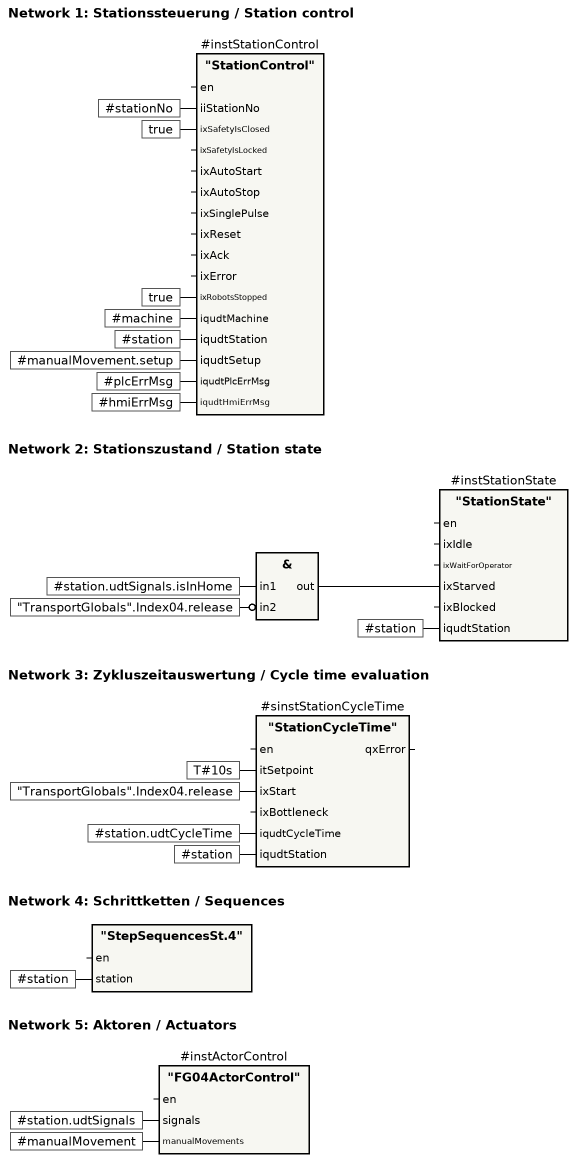
   #instStationControl(iiStationNo := #stationNo,   // "StationControl"
                       ixSafetyIsClosed := true,
                       ixRobotsStopped := true,
                       iqudtMachine := #machine,
                       iqudtStation := #station,
                       iqudtSetup := #manualMovement.setup,
                       iqudtPlcErrMsg := #plcErrMsg,
                       iqudtHmiErrMsg := #hmiErrMsg);
END_REGION

REGION Network 2: Stationszustand / Station state
   #instStationState(ixStarved := #station.udtSignals.isInHome AND NOT "TransportGlobals".Index04.release,   // "StationState"
                     iqudtStation := #station);
END_REGION

REGION Network 3: Zykluszeitauswertung / Cycle time evaluation
   #sinstStationCycleTime(itSetpoint := T#10s,   // "StationCycleTime"
                          ixStart := "TransportGlobals".Index04.release,
                          iqudtCycleTime := #station.udtCycleTime,
                          iqudtStation := #station);
END_REGION

REGION Network 4: Schrittketten / Sequences
   "StepSequencesSt.4"(station := #station);
END_REGION

REGION Network 5: Aktoren / Actuators
   #instActorControl(signals := #station.udtSignals, manualMovements := #manualMovement);   // "FG04ActorControl"
END_REGION
END_FUNCTION_BLOCK

FUNCTION_BLOCK "FG04ActorControl"   // FB1402, FBD
TITLE = Aktoransteuerung / Actuator control
{ S7_Optimized_Access := 'TRUE' }
VERSION : 0.1
// Ersteller: Andreas Fast Automation
// Kontakt per LinkedIn: https://www.linkedin.com/in/automation-fast-andreas/
// 
// Das Projekt dient zu Demonstrationszwecken und kann frei genutzt werden.
// 
// Bausteinbeschreibung:
// Author: Andreas Fast Automation
// Kontakt per LinkedIn: https://www.linkedin.com/in/automation-fast-andreas/
// 
// This project is intended for demonstration purposes and may be used freely.
// 
// Block description:
   VAR_IN_OUT
      signals : "typeStationSignals";
      manualMovements : "typeManualMovements";
   END_VAR
   VAR
      sinstActorReserved1 : "Actor_Reserved";
      sinstActorReserved2 : "Actor_Reserved";
      sinstActorReserved3 : "Actor_Reserved";
      sinstAxisZ : "Cylinder_2Out2In";
   END_VAR
BEGIN

REGION Network 1: Achse Z / Axis Z
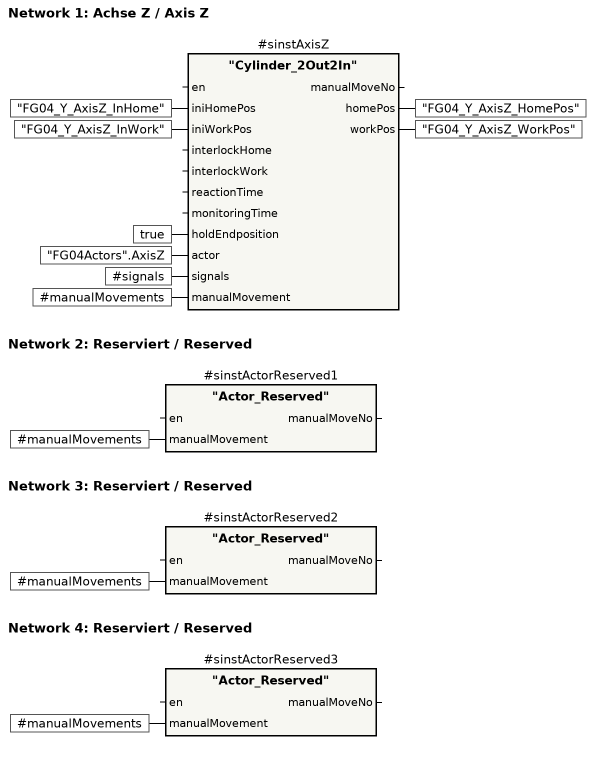
   #sinstAxisZ(iniHomePos := "FG04_Y_AxisZ_InHome",   // "Cylinder_2Out2In"
               iniWorkPos := "FG04_Y_AxisZ_InWork",
               holdEndposition := true,
               actor := "FG04Actors".AxisZ,
               signals := #signals,
               manualMovement := #manualMovements,
               homePos => "FG04_Y_AxisZ_HomePos",
               workPos => "FG04_Y_AxisZ_WorkPos");
END_REGION

REGION Network 2: Reserviert / Reserved
   #sinstActorReserved1(manualMovement := #manualMovements);   // "Actor_Reserved"
END_REGION

REGION Network 3: Reserviert / Reserved
   #sinstActorReserved2(manualMovement := #manualMovements);   // "Actor_Reserved"
END_REGION

REGION Network 4: Reserviert / Reserved
   #sinstActorReserved3(manualMovement := #manualMovements);   // "Actor_Reserved"
END_REGION
END_FUNCTION_BLOCK

// folder: 2. Machine/04_FG04/Stepsequences

